LIN {X 0,Y 499.621,Z 974.079,A -85,B 0,C 180,E1 -11819.006,E2 -11819.006} C_VEL
LIN {X 0,Y 503.101,Z 958.378,A -85,B 0,C 180,E1 -11821.283,E2 -11821.283} C_VEL
LIN {X 0,Y 506.634,Z 942.412,A -85,B 0,C 180,E1 -11823.275,E2 -11823.275} C_VEL
LIN {X 0,Y 510.604,Z 924.617,A -85,B 0,C 180,E1 -11825.226,E2 -11825.226} C_VEL
LIN {X 0,Y 514.669,Z 905.302,A -85,B 0,C 180,E1 -11827.032,E2 -11827.032} C_VEL
LIN {X 0,Y 518.595,Z 886.147,A -85,B 0,C 180,E1 -11828.589,E2 -11828.589} C_VEL
LIN {X 0,Y 522.625,Z 864.682,A -85,B 0,C 180,E1 -11830.067,E2 -11830.067} C_VEL
LIN {X 0,Y 525.92,Z 845.573,A -85,B 0,C 180,E1 -11831.195,E2 -11831.195} C_VEL
LIN {X 0,Y 529.613,Z 821.59,A -85,B 0,C 180,E1 -11832.377,E2 -11832.377} C_VEL
LIN {X 0,Y 532.123,Z 802.454,A -85,B 0,C 180,E1 -11833.155,E2 -11833.155} C_VEL
LIN {X 0,Y 534.743,Z 779.457,A -85,B 0,C 180,E1 -11833.92,E2 -11833.92} C_VEL
LIN {X 0,Y 536.744,Z 755.79,A -85,B 0,C 180,E1 -11834.509,E2 -11834.509} C_VEL
LIN {X 0,Y 538.049,Z 733.759,A -85,B 0,C 180,E1 -11834.915,E2 -11834.915} C_VEL
LIN {X 0,Y 547.283,Z 482.875,A -85,B 0,C 180,E1 -11838.589,E2 -11838.589} C_VEL
LIN {X 0,Y 548.708,Z 441.821,A -85,B 0,C 180,E1 -11839.21,E2 -11839.21} C_VEL
LIN {X 0,Y 535.529,Z 420.602,A -85,B 0,C 180,E1 -11841.248,E2 -11841.248} C_VEL
LIN {X 0,Y 523.411,Z 403.652,A -85,B 0,C 180,E1 -11843.243,E2 -11843.243} C_VEL
LIN {X 0,Y 511.927,Z 388.487,A -85,B 0,C 180,E1 -11845.295,E2 -11845.295} C_VEL
LIN {X 0,Y 507.19,Z 382.618,A -85,B 0,C 180,E1 -11846.19,E2 -11846.19} C_VEL
LIN {X 0,Y 503.446,Z 377.826,A -85,B 0,C 180,E1 -11846.929,E2 -11846.929} C_VEL
LIN {X 0,Y 500.235,Z 374.018,A -85,B 0,C 180,E1 -11847.575,E2 -11847.575} C_VEL
LIN {X 0,Y 498.921,Z 372.158,A -85,B 0,C 180,E1 -11847.853,E2 -11847.853} C_VEL
LIN {X 0,Y 495.879,Z 368.896,A -85,B 0,C 180,E1 -11848.483,E2 -11848.483} C_VEL
LIN {X 0,Y 494.405,Z 366.407,A -85,B 0,C 180,E1 -11848.819,E2 -11848.819} C_VEL
LIN {X 0,Y 491.612,Z 364.144,A -85,B 0,C 180,E1 -11849.404,E2 -11849.404} C_VEL
LIN {X 0,Y 490.187,Z 361.183,A -85,B 0,C 180,E1 -11849.758,E2 -11849.758} C_VEL
LIN {X 0,Y 490,Z 360.194,A -85,B 0,C 180,E1 -11849.835,E2 -11849.835} C_VEL
LIN {X 0,Y 489.946,Z 360.203,A -85,B 0,C 180,E1 -11853.191,E2 -11853.191} C_VEL
LIN {X 0,Y 489.937,Z 360.203,A -85,B 0,C 180,E1 -11856.803,E2 -11856.803} C_VEL
LIN {X 0,Y 489.981,Z 360.199,A -85,B 0,C 180,E1 -11860.199,E2 -11860.199} C_VEL
LIN {X 0,Y 489.973,Z 360.196,A -85,B 0,C 180,E1 -11863.765,E2 -11863.765} C_VEL
LIN {X 0,Y 489.933,Z 360.192,A -85,B 0,C 180,E1 -11867.147,E2 -11867.147} C_VEL
LIN {X 0,Y 489.954,Z 360.179,A -85,B 0,C 180,E1 -11870.604,E2 -11870.604} C_VEL
LIN {X 0,Y 489.968,Z 360.177,A -85,B 0,C 180,E1 -11873.908,E2 -11873.908} C_VEL
LIN {X 0,Y 489.934,Z 360.192,A -85,B 0,C 180,E1 -11877.427,E2 -11877.427} C_VEL
LIN {X 0,Y 489.94,Z 360.201,A -85,B 0,C 180,E1 -11881.052,E2 -11881.052} C_VEL
LIN {X 0,Y 489.979,Z 360.194,A -85,B 0,C 180,E1 -11884.565,E2 -11884.565} C_VEL
LIN {X 0,Y 489.951,Z 360.18,A -85,B 0,C 180,E1 -11887.977,E2 -11887.977} C_VEL
LIN {X 0,Y 489.93,Z 360.176,A -85,B 0,C 180,E1 -11891.418,E2 -11891.418} C_VEL
LIN {X 0,Y 489.964,Z 360.175,A -85,B 0,C 180,E1 -11894.9,E2 -11894.9} C_VEL
LIN {X 0,Y 489.974,Z 360.182,A -85,B 0,C 180,E1 -11898.391,E2 -11898.391} C_VEL
LIN {X 0,Y 489.933,Z 360.199,A -85,B 0,C 180,E1 -11901.804,E2 -11901.804} C_VEL
LIN {X 0,Y 489.943,Z 360.201,A -85,B 0,C 180,E1 -11905.377,E2 -11905.377} C_VEL
LIN {X 0,Y 489.992,Z 360.197,A -85,B 0,C 180,E1 -11908.923,E2 -11908.923} C_VEL
LIN {X 0,Y 490.017,Z 360.424,A -85,B 0,C 180,E1 -11910.673,E2 -11910.673} C_VEL
LIN {X 0,Y 491.418,Z 363.93,A -85,B 0,C 180,E1 -11911.528,E2 -11911.528} C_VEL
LIN {X 0,Y 492.392,Z 365.741,A -85,B 0,C 180,E1 -11912.006,E2 -11912.006} C_VEL
LIN {X 0,Y 494.518,Z 369.645,A -85,B 0,C 180,E1 -11912.954,E2 -11912.954} C_VEL
LIN {X 0,Y 497.801,Z 374.223,A -85,B 0,C 180,E1 -11913.668,E2 -11913.668} C_VEL
LIN {X 0,Y 507.638,Z 387.39,A -85,B 0,C 180,E1 -11915.664,E2 -11915.664} C_VEL
LIN {X 0,Y 516.631,Z 399.971,A -85,B 0,C 180,E1 -11917.355,E2 -11917.355} C_VEL
LIN {X 0,Y 527.787,Z 416.461,A -85,B 0,C 180,E1 -11919.307,E2 -11919.307} C_VEL
LIN {X 0,Y 540.338,Z 436.58,A -85,B 0,C 180,E1 -11921.348,E2 -11921.348} C_VEL
LIN {X 0,Y 548.723,Z 451.311,A -85,B 0,C 180,E1 -11922.64,E2 -11922.64} C_VEL
LIN {X 0,Y 539.479,Z 702.482,A -85,B 0,C 180,E1 -11926.318,E2 -11926.318} C_VEL
LIN {X 0,Y 537.078,Z 765.181,A -85,B 0,C 180,E1 -11927.257,E2 -11927.257} C_VEL
LIN {X 0,Y 535.059,Z 790.28,A -85,B 0,C 180,E1 -11927.793,E2 -11927.793} C_VEL
LIN {X 0,Y 532.837,Z 811.473,A -85,B 0,C 180,E1 -11928.394,E2 -11928.394} C_VEL
LIN {X 0,Y 529.672,Z 836.124,A -85,B 0,C 180,E1 -11929.291,E2 -11929.291} C_VEL
LIN {X 0,Y 526.628,Z 856.667,A -85,B 0,C 180,E1 -11930.219,E2 -11930.219} C_VEL
LIN {X 0,Y 522.863,Z 879.253,A -85,B 0,C 180,E1 -11931.434,E2 -11931.434} C_VEL
LIN {X 0,Y 519.029,Z 900.032,A -85,B 0,C 180,E1 -11932.778,E2 -11932.778} C_VEL
LIN {X 0,Y 515.052,Z 920.507,A -85,B 0,C 180,E1 -11934.312,E2 -11934.312} C_VEL
LIN {X 0,Y 510.952,Z 940.064,A -85,B 0,C 180,E1 -11936.041,E2 -11936.041} C_VEL
LIN {X 0,Y 507.093,Z 958.257,A -85,B 0,C 180,E1 -11937.879,E2 -11937.879} C_VEL
LIN {X 0,Y 503.262,Z 975.902,A -85,B 0,C 180,E1 -11939.955,E2 -11939.955} C_VEL
LIN {X 0,Y 499.916,Z 991.806,A -85,B 0,C 180,E1 -11942.094,E2 -11942.094} C_VEL
LIN {X 0,Y 496.763,Z 1007.17,A -85,B 0,C 180,E1 -11944.485,E2 -11944.485} C_VEL
LIN {X 0,Y 494.443,Z 1019.312,A -85,B 0,C 180,E1 -11946.651,E2 -11946.651} C_VEL
LIN {X 0,Y 492.101,Z 1032.754,A -85,B 0,C 180,E1 -11949.42,E2 -11949.42} C_VEL
LIN {X 0,Y 490.58,Z 1042.696,A -85,B 0,C 180,E1 -11951.83,E2 -11951.83} C_VEL
LIN {X 0,Y 489.408,Z 1052.094,A -85,B 0,C 180,E1 -11954.476,E2 -11954.476} C_VEL
LIN {X 0,Y 488.611,Z 1060.001,A -85,B 0,C 180,E1 -11957.232,E2 -11957.232} C_VEL
LIN {X 0,Y 488.21,Z 1065.616,A -85,B 0,C 180,E1 -11959.617,E2 -11959.617} C_VEL
LIN {X 0,Y 487.988,Z 1070.959,A -85,B 0,C 180,E1 -11962.583,E2 -11962.583} C_VEL
LIN {X 0,Y 487.94,Z 1074.004,A -85,B 0,C 180,E1 -11965.063,E2 -11965.063} C_VEL
LIN {X 0,Y 487.927,Z 1075.86,A -85,B 0,C 180,E1 -11967.534,E2 -11967.534} C_VEL
LIN {X 0,Y 487.924,Z 1076.467,A -85,B 0,C 180,E1 -11970.352,E2 -11970.352} C_VEL
LIN {X 0,Y 487.93,Z 1075.637,A -85,B 0,C 180,E1 -11972.819,E2 -11972.819} C_VEL
LIN {X 0,Y 487.941,Z 1073.628,A -85,B 0,C 180,E1 -11975.291,E2 -11975.291} C_VEL
LIN {X 0,Y 488.035,Z 1069.53,A -85,B 0,C 180,E1 -11978.279,E2 -11978.279} C_VEL
LIN {X 0,Y 488.264,Z 1064.748,A -85,B 0,C 180,E1 -11980.74,E2 -11980.74} C_VEL
LIN {X 0,Y 488.784,Z 1058.014,A -85,B 0,C 180,E1 -11983.486,E2 -11983.486} C_VEL
LIN {X 0,Y 489.667,Z 1049.398,A -85,B 0,C 180,E1 -11986.245,E2 -11986.245} C_VEL
LIN {X 0,Y 490.902,Z 1040.057,A -85,B 0,C 180,E1 -11988.773,E2 -11988.773} C_VEL
LIN {X 0,Y 492.69,Z 1028.406,A -85,B 0,C 180,E1 -11991.426,E2 -11991.426} C_VEL
LIN {X 0,Y 494.724,Z 1016.75,A -85,B 0,C 180,E1 -11993.716,E2 -11993.716} C_VEL
LIN {X 0,Y 497.688,Z 1001.146,A -85,B 0,C 180,E1 -11996.36,E2 -11996.36} C_VEL
LIN {X 0,Y 500.61,Z 986.526,A -85,B 0,C 180,E1 -11998.498,E2 -11998.498} C_VEL
LIN {X 0,Y 504.41,Z 968.165,A -85,B 0,C 180,E1 -12000.825,E2 -12000.825} C_VEL
LIN {X 0,Y 507.711,Z 952.169,A -85,B 0,C 180,E1 -12002.584,E2 -12002.584} C_VEL
LIN {X 0,Y 511.658,Z 932.877,A -85,B 0,C 180,E1 -12004.443,E2 -12004.443} C_VEL
LIN {X 0,Y 515.488,Z 913.172,A -85,B 0,C 180,E1 -12006.065,E2 -12006.065} C_VEL
LIN {X 0,Y 519.375,Z 892.502,A -85,B 0,C 180,E1 -12007.54,E2 -12007.54} C_VEL
LIN {X 0,Y 522.872,Z 871.802,A -85,B 0,C 180,E1 -12008.782,E2 -12008.782} C_VEL
LIN {X 0,Y 525.902,Z 852.464,A -85,B 0,C 180,E1 -12009.776,E2 -12009.776} C_VEL
LIN {X 0,Y 529.266,Z 827.978,A -85,B 0,C 180,E1 -12010.818,E2 -12010.818} C_VEL
LIN {X 0,Y 531.66,Z 807.467,A -85,B 0,C 180,E1 -12011.517,E2 -12011.517} C_VEL
LIN {X 0,Y 533.992,Z 783.772,A -85,B 0,C 180,E1 -12012.157,E2 -12012.157} C_VEL
LIN {X 0,Y 535.574,Z 759.261,A -85,B 0,C 180,E1 -12012.627,E2 -12012.627} C_VEL
LIN {X 0,Y 543.706,Z 523.272,A -85,B 0,C 180,E1 -12016.069,E2 -12016.069} C_VEL
LIN {X 0,Y 546.171,Z 449.822,A -85,B 0,C 180,E1 -12017.16,E2 -12017.16} C_VEL
LIN {X 0,Y 533.572,Z 427.973,A -85,B 0,C 180,E1 -12019.013,E2 -12019.013} C_VEL
LIN {X 0,Y 520.585,Z 407.244,A -85,B 0,C 180,E1 -12021.056,E2 -12021.056} C_VEL
LIN {X 0,Y 507.929,Z 388.602,A -85,B 0,C 180,E1 -12023.206,E2 -12023.206} C_VEL
LIN {X 0,Y 497.103,Z 373.702,A -85,B 0,C 180,E1 -12025.198,E2 -12025.198} C_VEL
LIN {X 0,Y 494.207,Z 369.566,A -85,B 0,C 180,E1 -12025.774,E2 -12025.774} C_VEL
LIN {X 0,Y 492.163,Z 365.3,A -85,B 0,C 180,E1 -12026.733,E2 -12026.733} C_VEL
LIN {X 0,Y 489.994,Z 360.56,A -85,B 0,C 180,E1 -12027.818,E2 -12027.818} C_VEL
LIN {X 0,Y 489.934,Z 360.191,A -85,B 0,C 180,E1 -12027.952,E2 -12027.952} C_VEL
LIN {X 0,Y 489.991,Z 360.186,A -85,B 0,C 180,E1 -12031.344,E2 -12031.344} C_VEL
LIN {X 0,Y 489.963,Z 360.198,A -85,B 0,C 180,E1 -12034.882,E2 -12034.882} C_VEL
LIN {X 0,Y 489.931,Z 360.197,A -85,B 0,C 180,E1 -12038.321,E2 -12038.321} C_VEL
LIN {X 0,Y 489.956,Z 360.176,A -85,B 0,C 180,E1 -12041.806,E2 -12041.806} C_VEL
LIN {X 0,Y 489.99,Z 360.167,A -85,B 0,C 180,E1 -12045.343,E2 -12045.343} C_VEL
LIN {X 0,Y 489.941,Z 360.196,A -85,B 0,C 180,E1 -12048.821,E2 -12048.821} C_VEL
LIN {X 0,Y 489.934,Z 360.198,A -85,B 0,C 180,E1 -12052.377,E2 -12052.377} C_VEL
LIN {X 0,Y 489.975,Z 360.165,A -85,B 0,C 180,E1 -12055.787,E2 -12055.787} C_VEL
LIN {X 0,Y 489.962,Z 360.184,A -85,B 0,C 180,E1 -12059.298,E2 -12059.298} C_VEL
LIN {X 0,Y 489.934,Z 360.201,A -85,B 0,C 180,E1 -12062.808,E2 -12062.808} C_VEL
LIN {X 0,Y 489.946,Z 360.169,A -85,B 0,C 180,E1 -12066.344,E2 -12066.344} C_VEL
LIN {X 0,Y 489.983,Z 360.18,A -85,B 0,C 180,E1 -12069.752,E2 -12069.752} C_VEL
LIN {X 0,Y 489.942,Z 360.199,A -85,B 0,C 180,E1 -12073.226,E2 -12073.226} C_VEL
LIN {X 0,Y 489.934,Z 360.176,A -85,B 0,C 180,E1 -12076.846,E2 -12076.846} C_VEL
LIN {X 0,Y 489.973,Z 360.171,A -85,B 0,C 180,E1 -12080.299,E2 -12080.299} C_VEL
LIN {X 0,Y 489.964,Z 360.195,A -85,B 0,C 180,E1 -12083.705,E2 -12083.705} C_VEL
LIN {X 0,Y 489.94,Z 360.202,A -85,B 0,C 180,E1 -12087.203,E2 -12087.203} C_VEL
LIN {X 0,Y 489.957,Z 360.186,A -85,B 0,C 180,E1 -12090.677,E2 -12090.677} C_VEL
LIN {X 0,Y 489.984,Z 360.179,A -85,B 0,C 180,E1 -12094.138,E2 -12094.138} C_VEL
LIN {X 0,Y 489.958,Z 360.256,A -85,B 0,C 180,E1 -12095.709,E2 -12095.709} C_VEL
LIN {X 0,Y 491.007,Z 363.245,A -85,B 0,C 180,E1 -12095.962,E2 -12095.962} C_VEL
LIN {X 0,Y 493.4,Z 365.788,A -85,B 0,C 180,E1 -12096.425,E2 -12096.425} C_VEL
LIN {X 0,Y 494.526,Z 366.796,A -85,B 0,C 180,E1 -12096.635,E2 -12096.635} C_VEL
LIN {X 0,Y 496.989,Z 370.604,A -85,B 0,C 180,E1 -12097.126,E2 -12097.126} C_VEL
LIN {X 0,Y 499.262,Z 372.917,A -85,B 0,C 180,E1 -12097.542,E2 -12097.542} C_VEL
LIN {X 0,Y 502.564,Z 377.233,A -85,B 0,C 180,E1 -12098.153,E2 -12098.153} C_VEL
LIN {X 0,Y 512.006,Z 389.56,A -85,B 0,C 180,E1 -12099.815,E2 -12099.815} C_VEL
LIN {X 0,Y 523.641,Z 405.343,A -85,B 0,C 180,E1 -12101.718,E2 -12101.718} C_VEL
LIN {X 0,Y 534.992,Z 421.994,A -85,B 0,C 180,E1 -12103.455,E2 -12103.455} C_VEL
LIN {X 0,Y 546.448,Z 441.202,A -85,B 0,C 180,E1 -12105.128,E2 -12105.128} C_VEL
LIN {X 0,Y 537.807,Z 687.67,A -85,B 0,C 180,E1 -12108.714,E2 -12108.714} C_VEL
LIN {X 0,Y 535.684,Z 744.725,A -85,B 0,C 180,E1 -12109.568,E2 -12109.568} C_VEL
LIN {X 0,Y 533.884,Z 769.233,A -85,B 0,C 180,E1 -12110.108,E2 -12110.108} C_VEL
LIN {X 0,Y 531.773,Z 791.218,A -85,B 0,C 180,E1 -12110.75,E2 -12110.75} C_VEL
LIN {X 0,Y 528.953,Z 814.971,A -85,B 0,C 180,E1 -12111.639,E2 -12111.639} C_VEL
LIN {X 0,Y 526.187,Z 834.834,A -85,B 0,C 180,E1 -12112.549,E2 -12112.549} C_VEL
LIN {X 0,Y 522.677,Z 857.192,A -85,B 0,C 180,E1 -12113.763,E2 -12113.763} C_VEL
LIN {X 0,Y 519.054,Z 877.695,A -85,B 0,C 180,E1 -12115.101,E2 -12115.101} C_VEL
LIN {X 0,Y 515.255,Z 897.885,A -85,B 0,C 180,E1 -12116.623,E2 -12116.623} C_VEL
LIN {X 0,Y 511.312,Z 917.088,A -85,B 0,C 180,E1 -12118.328,E2 -12118.328} C_VEL
LIN {X 0,Y 510.97,Z 918.726,A -85,B 0,C 180,E1 -12118.484,E2 -12118.484} C_VEL
LIN {X 0,Y 508.908,Z 924.702,A -85,B 0,C 180,E1 -12118.999,E2 -12118.999} C_VEL
LIN {X 0,Y 500.503,Z 939.528,A -85,B 0,C 180,E1 -12120.219,E2 -12120.219} C_VEL
LIN {X 0,Y 498.41,Z 944.959,A -85,B 0,C 180,E1 -12120.796,E2 -12120.796} C_VEL
LIN {X 0,Y 494.435,Z 962.729,A -85,B 0,C 180,E1 -12123.105,E2 -12123.105} C_VEL
LIN {X 0,Y 491.323,Z 976.784,A -85,B 0,C 180,E1 -12125.214,E2 -12125.214} C_VEL
LIN {X 0,Y 488.087,Z 992.002,A -85,B 0,C 180,E1 -12127.856,E2 -12127.856} C_VEL
LIN {X 0,Y 485.71,Z 1003.891,A -85,B 0,C 180,E1 -12130.269,E2 -12130.269} C_VEL
LIN {X 0,Y 483.54,Z 1016.07,A -85,B 0,C 180,E1 -12133.172,E2 -12133.172} C_VEL
LIN {X 0,Y 482.208,Z 1024.593,A -85,B 0,C 180,E1 -12135.592,E2 -12135.592} C_VEL
LIN {X 0,Y 481.157,Z 1032.862,A -85,B 0,C 180,E1 -12138.371,E2 -12138.371} C_VEL
LIN {X 0,Y 480.498,Z 1039.328,A -85,B 0,C 180,E1 -12141.142,E2 -12141.142} C_VEL
LIN {X 0,Y 480.163,Z 1043.981,A -85,B 0,C 180,E1 -12143.664,E2 -12143.664} C_VEL
LIN {X 0,Y 479.987,Z 1047.874,A -85,B 0,C 180,E1 -12146.656,E2 -12146.656} C_VEL
LIN {X 0,Y 479.945,Z 1049.749,A -85,B 0,C 180,E1 -12149.045,E2 -12149.045} C_VEL
LIN {X 0,Y 479.923,Z 1050.584,A -85,B 0,C 180,E1 -12151.433,E2 -12151.433} C_VEL
LIN {X 0,Y 479.94,Z 1050.138,A -85,B 0,C 180,E1 -12154.421,E2 -12154.421} C_VEL
LIN {X 0,Y 479.981,Z 1048.405,A -85,B 0,C 180,E1 -12156.94,E2 -12156.94} C_VEL
LIN {X 0,Y 480.088,Z 1045.678,A -85,B 0,C 180,E1 -12159.349,E2 -12159.349} C_VEL
LIN {X 0,Y 480.404,Z 1040.694,A -85,B 0,C 180,E1 -12162.379,E2 -12162.379} C_VEL
LIN {X 0,Y 480.947,Z 1035.03,A -85,B 0,C 180,E1 -12164.939,E2 -12164.939} C_VEL
LIN {X 0,Y 481.928,Z 1027.365,A -85,B 0,C 180,E1 -12167.763,E2 -12167.763} C_VEL
LIN {X 0,Y 483.383,Z 1017.776,A -85,B 0,C 180,E1 -12170.588,E2 -12170.588} C_VEL
LIN {X 0,Y 485.367,Z 1006.968,A -85,B 0,C 180,E1 -12173.299,E2 -12173.299} C_VEL
LIN {X 0,Y 487.847,Z 994.643,A -85,B 0,C 180,E1 -12175.885,E2 -12175.885} C_VEL
LIN {X 0,Y 490.638,Z 981.902,A -85,B 0,C 180,E1 -12178.216,E2 -12178.216} C_VEL
LIN {X 0,Y 494.168,Z 966.354,A -85,B 0,C 180,E1 -12180.657,E2 -12180.657} C_VEL
LIN {X 0,Y 497.539,Z 951.848,A -85,B 0,C 180,E1 -12182.642,E2 -12182.642} C_VEL
LIN {X 0,Y 501.913,Z 933.015,A -85,B 0,C 180,E1 -12184.872,E2 -12184.872} C_VEL
LIN {X 0,Y 505.593,Z 916.81,A -85,B 0,C 180,E1 -12186.532,E2 -12186.532} C_VEL
LIN {X 0,Y 509.926,Z 897.147,A -85,B 0,C 180,E1 -12188.289,E2 -12188.289} C_VEL
LIN {X 0,Y 513.894,Z 877.606,A -85,B 0,C 180,E1 -12189.775,E2 -12189.775} C_VEL
LIN {X 0,Y 517.938,Z 856.354,A -85,B 0,C 180,E1 -12191.171,E2 -12191.171} C_VEL
LIN {X 0,Y 521.615,Z 834.431,A -85,B 0,C 180,E1 -12192.361,E2 -12192.361} C_VEL
LIN {X 0,Y 524.717,Z 813.622,A -85,B 0,C 180,E1 -12193.315,E2 -12193.315} C_VEL
LIN {X 0,Y 527.783,Z 789.004,A -85,B 0,C 180,E1 -12194.22,E2 -12194.22} C_VEL
LIN {X 0,Y 530.012,Z 767.069,A -85,B 0,C 180,E1 -12194.85,E2 -12194.85} C_VEL
LIN {X 0,Y 531.932,Z 740.911,A -85,B 0,C 180,E1 -12195.396,E2 -12195.396} C_VEL
LIN {X 0,Y 540.8,Z 510.38,A -85,B 0,C 180,E1 -12198.811,E2 -12198.811} C_VEL
LIN {X 0,Y 543.236,Z 445.431,A -85,B 0,C 180,E1 -12199.789,E2 -12199.789} C_VEL
LIN {X 0,Y 530.888,Z 425.495,A -85,B 0,C 180,E1 -12201.752,E2 -12201.752} C_VEL
LIN {X 0,Y 519.483,Z 409.528,A -85,B 0,C 180,E1 -12203.676,E2 -12203.676} C_VEL
LIN {X 0,Y 508.649,Z 395.076,A -85,B 0,C 180,E1 -12205.655,E2 -12205.655} C_VEL
LIN {X 0,Y 503.459,Z 388.623,A -85,B 0,C 180,E1 -12206.658,E2 -12206.658} C_VEL
LIN {X 0,Y 500.253,Z 384.501,A -85,B 0,C 180,E1 -12207.305,E2 -12207.305} C_VEL
LIN {X 0,Y 496.742,Z 380.013,A -85,B 0,C 180,E1 -12208.035,E2 -12208.035} C_VEL
LIN {X 0,Y 492.563,Z 375.092,A -85,B 0,C 180,E1 -12208.927,E2 -12208.927} C_VEL
LIN {X 0,Y 491.539,Z 373.531,A -85,B 0,C 180,E1 -12209.161,E2 -12209.161} C_VEL
LIN {X 0,Y 488.465,Z 370.552,A -85,B 0,C 180,E1 -12209.832,E2 -12209.832} C_VEL
LIN {X 0,Y 486.735,Z 367.519,A -85,B 0,C 180,E1 -12210.257,E2 -12210.257} C_VEL
LIN {X 0,Y 483.812,Z 365.336,A -85,B 0,C 180,E1 -12210.909,E2 -12210.909} C_VEL
LIN {X 0,Y 482.264,Z 362.395,A -85,B 0,C 180,E1 -12211.316,E2 -12211.316} C_VEL
LIN {X 0,Y 482.022,Z 361.171,A -85,B 0,C 180,E1 -12211.425,E2 -12211.425} C_VEL
LIN {X 0,Y 481.997,Z 361.171,A -85,B 0,C 180,E1 -12214.963,E2 -12214.963} C_VEL
LIN {X 0,Y 482.013,Z 361.168,A -85,B 0,C 180,E1 -12218.459,E2 -12218.459} C_VEL
LIN {X 0,Y 482.042,Z 361.165,A -85,B 0,C 180,E1 -12221.872,E2 -12221.872} C_VEL
LIN {X 0,Y 481.999,Z 361.173,A -85,B 0,C 180,E1 -12225.34,E2 -12225.34} C_VEL
LIN {X 0,Y 482,Z 361.182,A -85,B 0,C 180,E1 -12228.879,E2 -12228.879} C_VEL
LIN {X 0,Y 482.043,Z 361.186,A -85,B 0,C 180,E1 -12232.371,E2 -12232.371} C_VEL
LIN {X 0,Y 482.029,Z 361.182,A -85,B 0,C 180,E1 -12235.956,E2 -12235.956} C_VEL
LIN {X 0,Y 481.993,Z 361.172,A -85,B 0,C 180,E1 -12239.406,E2 -12239.406} C_VEL
LIN {X 0,Y 482.002,Z 361.165,A -85,B 0,C 180,E1 -12242.973,E2 -12242.973} C_VEL
LIN {X 0,Y 482.05,Z 361.162,A -85,B 0,C 180,E1 -12246.504,E2 -12246.504} C_VEL
LIN {X 0,Y 482.015,Z 361.178,A -85,B 0,C 180,E1 -12250.035,E2 -12250.035} C_VEL
LIN {X 0,Y 481.994,Z 361.191,A -85,B 0,C 180,E1 -12253.557,E2 -12253.557} C_VEL
LIN {X 0,Y 482.02,Z 361.181,A -85,B 0,C 180,E1 -12257.007,E2 -12257.007} C_VEL
LIN {X 0,Y 482.042,Z 361.168,A -85,B 0,C 180,E1 -12260.521,E2 -12260.521} C_VEL
LIN {X 0,Y 481.994,Z 361.168,A -85,B 0,C 180,E1 -12263.862,E2 -12263.862} C_VEL
LIN {X 0,Y 482.002,Z 361.168,A -85,B 0,C 180,E1 -12267.421,E2 -12267.421} C_VEL
LIN {X 0,Y 482.039,Z 361.318,A -85,B 0,C 180,E1 -12269.208,E2 -12269.208} C_VEL
LIN {X 0,Y 483.265,Z 364.613,A -85,B 0,C 180,E1 -12270.047,E2 -12270.047} C_VEL
LIN {X 0,Y 484.518,Z 366.617,A -85,B 0,C 180,E1 -12270.646,E2 -12270.646} C_VEL
LIN {X 0,Y 485.699,Z 369.227,A -85,B 0,C 180,E1 -12271.251,E2 -12271.251} C_VEL
LIN {X 0,Y 491.205,Z 375.925,A -85,B 0,C 180,E1 -12272.507,E2 -12272.507} C_VEL
LIN {X 0,Y 495.053,Z 381.243,A -85,B 0,C 180,E1 -12273.359,E2 -12273.359} C_VEL
LIN {X 0,Y 506.429,Z 396.637,A -85,B 0,C 180,E1 -12275.693,E2 -12275.693} C_VEL
LIN {X 0,Y 516.502,Z 411.273,A -85,B 0,C 180,E1 -12277.593,E2 -12277.593} C_VEL
LIN {X 0,Y 527.061,Z 427.405,A -85,B 0,C 180,E1 -12279.442,E2 -12279.442} C_VEL
LIN {X 0,Y 538.473,Z 446.211,A -85,B 0,C 180,E1 -12281.31,E2 -12281.31} C_VEL
LIN {X 0,Y 543.243,Z 454.931,A -85,B 0,C 180,E1 -12282.064,E2 -12282.064} C_VEL
LIN {X 0,Y 533.685,Z 704.84,A -85,B 0,C 180,E1 -12285.751,E2 -12285.751} C_VEL
LIN {X 0,Y 531.274,Z 765.234,A -85,B 0,C 180,E1 -12286.664,E2 -12286.664} C_VEL
LIN {X 0,Y 529.199,Z 790.162,A -85,B 0,C 180,E1 -12287.201,E2 -12287.201} C_VEL
LIN {X 0,Y 526.93,Z 811.121,A -85,B 0,C 180,E1 -12287.798,E2 -12287.798} C_VEL
LIN {X 0,Y 523.593,Z 836.206,A -85,B 0,C 180,E1 -12288.716,E2 -12288.716} C_VEL
LIN {X 0,Y 520.443,Z 856.712,A -85,B 0,C 180,E1 -12289.65,E2 -12289.65} C_VEL
LIN {X 0,Y 516.41,Z 879.898,A -85,B 0,C 180,E1 -12290.912,E2 -12290.912} C_VEL
LIN {X 0,Y 512.556,Z 900,A -85,B 0,C 180,E1 -12292.226,E2 -12292.226} C_VEL
LIN {X 0,Y 508.269,Z 921.119,A -85,B 0,C 180,E1 -12293.831,E2 -12293.831} C_VEL
LIN {X 0,Y 504.207,Z 939.745,A -85,B 0,C 180,E1 -12295.496,E2 -12295.496} C_VEL
LIN {X 0,Y 500.318,Z 957.3,A -85,B 0,C 180,E1 -12297.286,E2 -12297.286} C_VEL
LIN {X 0,Y 496.118,Z 975.783,A -85,B 0,C 180,E1 -12299.477,E2 -12299.477} C_VEL
LIN {X 0,Y 492.794,Z 990.826,A -85,B 0,C 180,E1 -12301.522,E2 -12301.522} C_VEL
LIN {X 0,Y 489.298,Z 1007.022,A -85,B 0,C 180,E1 -12304.067,E2 -12304.067} C_VEL
LIN {X 0,Y 486.851,Z 1019.146,A -85,B 0,C 180,E1 -12306.263,E2 -12306.263} C_VEL
LIN {X 0,Y 484.368,Z 1032.585,A -85,B 0,C 180,E1 -12309.076,E2 -12309.076} C_VEL
LIN {X 0,Y 482.744,Z 1042.645,A -85,B 0,C 180,E1 -12311.558,E2 -12311.558} C_VEL
LIN {X 0,Y 481.465,Z 1052.283,A -85,B 0,C 180,E1 -12314.337,E2 -12314.337} C_VEL
LIN {X 0,Y 480.662,Z 1059.81,A -85,B 0,C 180,E1 -12317.017,E2 -12317.017} C_VEL
LIN {X 0,Y 480.236,Z 1065.421,A -85,B 0,C 180,E1 -12319.442,E2 -12319.442} C_VEL
LIN {X 0,Y 479.987,Z 1070.757,A -85,B 0,C 180,E1 -12322.459,E2 -12322.459} C_VEL
LIN {X 0,Y 479.941,Z 1073.798,A -85,B 0,C 180,E1 -12324.98,E2 -12324.98} C_VEL
LIN {X 0,Y 479.929,Z 1075.652,A -85,B 0,C 180,E1 -12327.492,E2 -12327.492} C_VEL
LIN {X 0,Y 479.927,Z 1076.252,A -85,B 0,C 180,E1 -12330.358,E2 -12330.358} C_VEL
LIN {X 0,Y 479.932,Z 1075.418,A -85,B 0,C 180,E1 -12332.866,E2 -12332.866} C_VEL
LIN {X 0,Y 479.942,Z 1073.521,A -85,B 0,C 180,E1 -12335.26,E2 -12335.26} C_VEL
LIN {X 0,Y 480.021,Z 1069.777,A -85,B 0,C 180,E1 -12338.143,E2 -12338.143} C_VEL
LIN {X 0,Y 480.272,Z 1064.769,A -85,B 0,C 180,E1 -12340.799,E2 -12340.799} C_VEL
LIN {X 0,Y 480.779,Z 1058.388,A -85,B 0,C 180,E1 -12343.47,E2 -12343.47} C_VEL
LIN {X 0,Y 481.734,Z 1049.553,A -85,B 0,C 180,E1 -12346.396,E2 -12346.396} C_VEL
LIN {X 0,Y 482.981,Z 1040.525,A -85,B 0,C 180,E1 -12348.896,E2 -12348.896} C_VEL
LIN {X 0,Y 484.994,Z 1028.127,A -85,B 0,C 180,E1 -12351.783,E2 -12351.783} C_VEL
LIN {X 0,Y 487.133,Z 1016.462,A -85,B 0,C 180,E1 -12354.109,E2 -12354.109} C_VEL
LIN {X 0,Y 490.255,Z 1000.843,A -85,B 0,C 180,E1 -12356.791,E2 -12356.791} C_VEL
LIN {X 0,Y 493.157,Z 986.966,A -85,B 0,C 180,E1 -12358.852,E2 -12358.852} C_VEL
LIN {X 0,Y 496.98,Z 969.373,A -85,B 0,C 180,E1 -12361.136,E2 -12361.136} C_VEL
LIN {X 0,Y 500.64,Z 952.33,A -85,B 0,C 180,E1 -12363.041,E2 -12363.041} C_VEL
LIN {X 0,Y 504.753,Z 933.076,A -85,B 0,C 180,E1 -12364.924,E2 -12364.924} C_VEL
LIN {X 0,Y 508.709,Z 913.527,A -85,B 0,C 180,E1 -12366.553,E2 -12366.553} C_VEL
LIN {X 0,Y 512.731,Z 892.926,A -85,B 0,C 180,E1 -12368.042,E2 -12368.042} C_VEL
LIN {X 0,Y 516.511,Z 871.435,A -85,B 0,C 180,E1 -12369.345,E2 -12369.345} C_VEL
LIN {X 0,Y 519.735,Z 851.531,A -85,B 0,C 180,E1 -12370.373,E2 -12370.373} C_VEL
LIN {X 0,Y 523.141,Z 827.416,A -85,B 0,C 180,E1 -12371.4,E2 -12371.4} C_VEL
LIN {X 0,Y 525.598,Z 807.062,A -85,B 0,C 180,E1 -12372.096,E2 -12372.096} C_VEL
LIN {X 0,Y 527.992,Z 783.427,A -85,B 0,C 180,E1 -12372.736,E2 -12372.736} C_VEL
LIN {X 0,Y 529.62,Z 758.915,A -85,B 0,C 180,E1 -12373.208,E2 -12373.208} C_VEL
LIN {X 0,Y 538.1,Z 522.435,A -85,B 0,C 180,E1 -12376.686,E2 -12376.686} C_VEL
LIN {X 0,Y 540.511,Z 453.255,A -85,B 0,C 180,E1 -12377.722,E2 -12377.722} C_VEL
LIN {X 0,Y 528.792,Z 432.769,A -85,B 0,C 180,E1 -12379.494,E2 -12379.494} C_VEL
LIN {X 0,Y 515.955,Z 412.163,A -85,B 0,C 180,E1 -12381.567,E2 -12381.567} C_VEL
LIN {X 0,Y 504.122,Z 394.665,A -85,B 0,C 180,E1 -12383.626,E2 -12383.626} C_VEL
LIN {X 0,Y 493.941,Z 380.422,A -85,B 0,C 180,E1 -12385.542,E2 -12385.542} C_VEL
LIN {X 0,Y 489.755,Z 374.884,A -85,B 0,C 180,E1 -12386.373,E2 -12386.373} C_VEL
LIN {X 0,Y 485.508,Z 369.065,A -85,B 0,C 180,E1 -12387.275,E2 -12387.275} C_VEL
LIN {X 0,Y 483.704,Z 365.21,A -85,B 0,C 180,E1 -12388.188,E2 -12388.188} C_VEL
LIN {X 0,Y 482.252,Z 362.279,A -85,B 0,C 180,E1 -12388.917,E2 -12388.917} C_VEL
LIN {X 0,Y 482.057,Z 361.159,A -85,B 0,C 180,E1 -12389.181,E2 -12389.181} C_VEL
LIN {X 0,Y 482.002,Z 361.162,A -85,B 0,C 180,E1 -12392.606,E2 -12392.606} C_VEL
LIN {X 0,Y 481.992,Z 361.164,A -85,B 0,C 180,E1 -12396.185,E2 -12396.185} C_VEL
LIN {X 0,Y 482.029,Z 361.175,A -85,B 0,C 180,E1 -12399.652,E2 -12399.652} C_VEL
LIN {X 0,Y 482.042,Z 361.186,A -85,B 0,C 180,E1 -12403.242,E2 -12403.242} C_VEL
LIN {X 0,Y 481.996,Z 361.17,A -85,B 0,C 180,E1 -12406.687,E2 -12406.687} C_VEL
LIN {X 0,Y 481.994,Z 361.158,A -85,B 0,C 180,E1 -12410.326,E2 -12410.326} C_VEL
LIN {X 0,Y 482.038,Z 361.178,A -85,B 0,C 180,E1 -12413.808,E2 -12413.808} C_VEL
LIN {X 0,Y 482.031,Z 361.179,A -85,B 0,C 180,E1 -12417.384,E2 -12417.384} C_VEL
LIN {X 0,Y 481.991,Z 361.155,A -85,B 0,C 180,E1 -12420.832,E2 -12420.832} C_VEL
LIN {X 0,Y 482.005,Z 361.18,A -85,B 0,C 180,E1 -12424.402,E2 -12424.402} C_VEL
LIN {X 0,Y 482.055,Z 361.176,A -85,B 0,C 180,E1 -12427.868,E2 -12427.868} C_VEL
LIN {X 0,Y 482.018,Z 361.154,A -85,B 0,C 180,E1 -12431.487,E2 -12431.487} C_VEL
LIN {X 0,Y 481.995,Z 361.175,A -85,B 0,C 180,E1 -12434.906,E2 -12434.906} C_VEL
LIN {X 0,Y 482.028,Z 361.188,A -85,B 0,C 180,E1 -12438.379,E2 -12438.379} C_VEL
LIN {X 0,Y 482.055,Z 361.164,A -85,B 0,C 180,E1 -12442.001,E2 -12442.001} C_VEL
LIN {X 0,Y 482.009,Z 361.16,A -85,B 0,C 180,E1 -12445.562,E2 -12445.562} C_VEL
LIN {X 0,Y 482,Z 361.166,A -85,B 0,C 180,E1 -12449.04,E2 -12449.04} C_VEL
LIN {X 0,Y 482.038,Z 361.169,A -85,B 0,C 180,E1 -12452.496,E2 -12452.496} C_VEL
LIN {X 0,Y 482.072,Z 361.362,A -85,B 0,C 180,E1 -12454.345,E2 -12454.345} C_VEL
LIN {X 0,Y 483.137,Z 364.357,A -85,B 0,C 180,E1 -12454.618,E2 -12454.618} C_VEL
LIN {X 0,Y 485.642,Z 366.951,A -85,B 0,C 180,E1 -12455.132,E2 -12455.132} C_VEL
LIN {X 0,Y 486.744,Z 367.867,A -85,B 0,C 180,E1 -12455.349,E2 -12455.349} C_VEL
LIN {X 0,Y 489.116,Z 371.544,A -85,B 0,C 180,E1 -12455.852,E2 -12455.852} C_VEL
LIN {X 0,Y 491.447,Z 373.923,A -85,B 0,C 180,E1 -12456.304,E2 -12456.304} C_VEL
LIN {X 0,Y 494.642,Z 378.163,A -85,B 0,C 180,E1 -12456.933,E2 -12456.933} C_VEL
LIN {X 0,Y 496.343,Z 380.199,A -85,B 0,C 180,E1 -12457.255,E2 -12457.255} C_VEL
LIN {X 0,Y 501.344,Z 386.76,A -85,B 0,C 180,E1 -12458.19,E2 -12458.19} C_VEL
LIN {X 0,Y 505.654,Z 392.322,A -85,B 0,C 180,E1 -12458.963,E2 -12458.963} C_VEL
LIN {X 0,Y 515.74,Z 405.857,A -85,B 0,C 180,E1 -12460.686,E2 -12460.686} C_VEL
LIN {X 0,Y 527.75,Z 423.031,A -85,B 0,C 180,E1 -12462.599,E2 -12462.599} C_VEL
LIN {X 0,Y 539.534,Z 442.323,A -85,B 0,C 180,E1 -12464.377,E2 -12464.377} C_VEL
LIN {X 0,Y 540.795,Z 444.867,A -85,B 0,C 180,E1 -12464.568,E2 -12464.568} C_VEL
LIN {X 0,Y 531.788,Z 692,A -85,B 0,C 180,E1 -12468.192,E2 -12468.192} C_VEL
LIN {X 0,Y 529.701,Z 745.554,A -85,B 0,C 180,E1 -12469.003,E2 -12469.003} C_VEL
LIN {X 0,Y 527.831,Z 769.887,A -85,B 0,C 180,E1 -12469.548,E2 -12469.548} C_VEL
LIN {X 0,Y 525.596,Z 792.386,A -85,B 0,C 180,E1 -12470.213,E2 -12470.213} C_VEL
LIN {X 0,Y 522.608,Z 816.404,A -85,B 0,C 180,E1 -12471.13,E2 -12471.13} C_VEL
LIN {X 0,Y 519.646,Z 836.867,A -85,B 0,C 180,E1 -12472.084,E2 -12472.084} C_VEL
LIN {X 0,Y 515.736,Z 860.378,A -85,B 0,C 180,E1 -12473.404,E2 -12473.404} C_VEL
LIN {X 0,Y 512.213,Z 879.579,A -85,B 0,C 180,E1 -12474.685,E2 -12474.685} C_VEL
LIN {X 0,Y 507.952,Z 900.99,A -85,B 0,C 180,E1 -12476.35,E2 -12476.35} C_VEL
LIN {X 0,Y 504.181,Z 918.716,A -85,B 0,C 180,E1 -12477.96,E2 -12477.96} C_VEL
LIN {X 0,Y 500.171,Z 937.19,A -85,B 0,C 180,E1 -12479.883,E2 -12479.883} C_VEL
LIN {X 0,Y 498.41,Z 944.959,A -85,B 0,C 180,E1 -12480.796,E2 -12480.796} C_VEL
LIN {X 0,Y 496.317,Z 950.385,A -85,B 0,C 180,E1 -12481.393,E2 -12481.393} C_VEL
LIN {X 0,Y 487.897,Z 963.83,A -85,B 0,C 180,E1 -12482.837,E2 -12482.837} C_VEL
LIN {X 0,Y 485.877,Z 968.772,A -85,B 0,C 180,E1 -12483.495,E2 -12483.495} C_VEL
LIN {X 0,Y 482.467,Z 983.638,A -85,B 0,C 180,E1 -12485.904,E2 -12485.904} C_VEL
LIN {X 0,Y 479.877,Z 995.452,A -85,B 0,C 180,E1 -12488.101,E2 -12488.101} C_VEL
LIN {X 0,Y 477.214,Z 1008.531,A -85,B 0,C 180,E1 -12490.922,E2 -12490.922} C_VEL
LIN {X 0,Y 475.439,Z 1018.17,A -85,B 0,C 180,E1 -12493.38,E2 -12493.38} C_VEL
LIN {X 0,Y 473.969,Z 1027.637,A -85,B 0,C 180,E1 -12496.209,E2 -12496.209} C_VEL
LIN {X 0,Y 472.98,Z 1035.212,A -85,B 0,C 180,E1 -12499.032,E2 -12499.032} C_VEL
LIN {X 0,Y 472.403,Z 1041.087,A -85,B 0,C 180,E1 -12501.725,E2 -12501.725} C_VEL
LIN {X 0,Y 472.095,Z 1045.818,A -85,B 0,C 180,E1 -12504.653,E2 -12504.653} C_VEL
LIN {X 0,Y 471.981,Z 1048.666,A -85,B 0,C 180,E1 -12507.207,E2 -12507.207} C_VEL
LIN {X 0,Y 471.951,Z 1050.529,A -85,B 0,C 180,E1 -12510.036,E2 -12510.036} C_VEL
LIN {X 0,Y 471.933,Z 1050.767,A -85,B 0,C 180,E1 -12512.915,E2 -12512.915} C_VEL
LIN {X 0,Y 471.954,Z 1049.871,A -85,B 0,C 180,E1 -12515.349,E2 -12515.349} C_VEL
LIN {X 0,Y 472.044,Z 1047.586,A -85,B 0,C 180,E1 -12518.159,E2 -12518.159} C_VEL
LIN {X 0,Y 472.23,Z 1043.669,A -85,B 0,C 180,E1 -12520.986,E2 -12520.986} C_VEL
LIN {X 0,Y 472.641,Z 1038.856,A -85,B 0,C 180,E1 -12523.581,E2 -12523.581} C_VEL
LIN {X 0,Y 473.523,Z 1031.375,A -85,B 0,C 180,E1 -12526.689,E2 -12526.689} C_VEL
LIN {X 0,Y 474.623,Z 1023.93,A -85,B 0,C 180,E1 -12529.187,E2 -12529.187} C_VEL
LIN {X 0,Y 476.439,Z 1013.732,A -85,B 0,C 180,E1 -12532.065,E2 -12532.065} C_VEL
LIN {X 0,Y 478.686,Z 1002.549,A -85,B 0,C 180,E1 -12534.694,E2 -12534.694} C_VEL
LIN {X 0,Y 481.571,Z 989.664,A -85,B 0,C 180,E1 -12537.314,E2 -12537.314} C_VEL
LIN {X 0,Y 484.842,Z 975.551,A -85,B 0,C 180,E1 -12539.746,E2 -12539.746} C_VEL
LIN {X 0,Y 488.67,Z 959.912,A -85,B 0,C 180,E1 -12542.101,E2 -12542.101} C_VEL
LIN {X 0,Y 492.747,Z 942.996,A -85,B 0,C 180,E1 -12544.271,E2 -12544.271} C_VEL
LIN {X 0,Y 497.039,Z 925.273,A -85,B 0,C 180,E1 -12546.259,E2 -12546.259} C_VEL
LIN {X 0,Y 501.465,Z 905.971,A -85,B 0,C 180,E1 -12548.103,E2 -12548.103} C_VEL
LIN {X 0,Y 505.714,Z 886.807,A -85,B 0,C 180,E1 -12549.69,E2 -12549.69} C_VEL
LIN {X 0,Y 510.061,Z 865.297,A -85,B 0,C 180,E1 -12551.199,E2 -12551.199} C_VEL
LIN {X 0,Y 513.423,Z 847.177,A -85,B 0,C 180,E1 -12552.288,E2 -12552.288} C_VEL
LIN {X 0,Y 517.343,Z 823.726,A -85,B 0,C 180,E1 -12553.476,E2 -12553.476} C_VEL
LIN {X 0,Y 520.212,Z 803.366,A -85,B 0,C 180,E1 -12554.321,E2 -12554.321} C_VEL
LIN {X 0,Y 522.826,Z 781.873,A -85,B 0,C 180,E1 -12555.051,E2 -12555.051} C_VEL
LIN {X 0,Y 525.117,Z 757.355,A -85,B 0,C 180,E1 -12555.684,E2 -12555.684} C_VEL
LIN {X 0,Y 526.51,Z 735.76,A -85,B 0,C 180,E1 -12556.093,E2 -12556.093} C_VEL
LIN {X 0,Y 536.423,Z 486.99,A -85,B 0,C 180,E1 -12559.793,E2 -12559.793} C_VEL
LIN {X 0,Y 537.887,Z 449.193,A -85,B 0,C 180,E1 -12560.369,E2 -12560.369} C_VEL
LIN {X 0,Y 526.627,Z 430.909,A -85,B 0,C 180,E1 -12562.208,E2 -12562.208} C_VEL
LIN {X 0,Y 515.323,Z 415.027,A -85,B 0,C 180,E1 -12564.162,E2 -12564.162} C_VEL
LIN {X 0,Y 505.137,Z 401.359,A -85,B 0,C 180,E1 -12566.068,E2 -12566.068} C_VEL
LIN {X 0,Y 497.21,Z 391.268,A -85,B 0,C 180,E1 -12567.661,E2 -12567.661} C_VEL
LIN {X 0,Y 492.535,Z 385.487,A -85,B 0,C 180,E1 -12568.653,E2 -12568.653} C_VEL
LIN {X 0,Y 489.056,Z 380.901,A -85,B 0,C 180,E1 -12569.431,E2 -12569.431} C_VEL
LIN {X 0,Y 485.457,Z 377.109,A -85,B 0,C 180,E1 -12570.239,E2 -12570.239} C_VEL
LIN {X 0,Y 483.938,Z 374.706,A -85,B 0,C 180,E1 -12570.612,E2 -12570.612} C_VEL
LIN {X 0,Y 480.759,Z 371.783,A -85,B 0,C 180,E1 -12571.354,E2 -12571.354} C_VEL
LIN {X 0,Y 478.908,Z 368.519,A -85,B 0,C 180,E1 -12571.845,E2 -12571.845} C_VEL
LIN {X 0,Y 475.901,Z 366.357,A -85,B 0,C 180,E1 -12572.57,E2 -12572.57} C_VEL
LIN {X 0,Y 474.353,Z 363.538,A -85,B 0,C 180,E1 -12573.008,E2 -12573.008} C_VEL
LIN {X 0,Y 474.067,Z 362.181,A -85,B 0,C 180,E1 -12573.148,E2 -12573.148} C_VEL
LIN {X 0,Y 474.061,Z 362.181,A -85,B 0,C 180,E1 -12576.77,E2 -12576.77} C_VEL
LIN {X 0,Y 474.095,Z 362.177,A -85,B 0,C 180,E1 -12580.278,E2 -12580.278} C_VEL
LIN {X 0,Y 474.101,Z 362.174,A -85,B 0,C 180,E1 -12583.836,E2 -12583.836} C_VEL
LIN {X 0,Y 474.06,Z 362.171,A -85,B 0,C 180,E1 -12587.329,E2 -12587.329} C_VEL
LIN {X 0,Y 474.056,Z 362.163,A -85,B 0,C 180,E1 -12591.02,E2 -12591.02} C_VEL
LIN {X 0,Y 474.095,Z 362.151,A -85,B 0,C 180,E1 -12594.433,E2 -12594.433} C_VEL
LIN {X 0,Y 474.085,Z 362.155,A -85,B 0,C 180,E1 -12597.945,E2 -12597.945} C_VEL
LIN {X 0,Y 474.057,Z 362.173,A -85,B 0,C 180,E1 -12601.45,E2 -12601.45} C_VEL
LIN {X 0,Y 474.063,Z 362.18,A -85,B 0,C 180,E1 -12605.082,E2 -12605.082} C_VEL
LIN {X 0,Y 474.103,Z 362.165,A -85,B 0,C 180,E1 -12608.612,E2 -12608.612} C_VEL
LIN {X 0,Y 474.084,Z 362.154,A -85,B 0,C 180,E1 -12612.176,E2 -12612.176} C_VEL
LIN {X 0,Y 474.053,Z 362.153,A -85,B 0,C 180,E1 -12615.663,E2 -12615.663} C_VEL
LIN {X 0,Y 474.065,Z 362.152,A -85,B 0,C 180,E1 -12619.21,E2 -12619.21} C_VEL
LIN {X 0,Y 474.119,Z 362.15,A -85,B 0,C 180,E1 -12622.702,E2 -12622.702} C_VEL
LIN {X 0,Y 474.078,Z 362.158,A -85,B 0,C 180,E1 -12626.314,E2 -12626.314} C_VEL
LIN {X 0,Y 474.077,Z 362.315,A -85,B 0,C 180,E1 -12627.646,E2 -12627.646} C_VEL
LIN {X 0,Y 475.302,Z 365.501,A -85,B 0,C 180,E1 -12628.525,E2 -12628.525} C_VEL
LIN {X 0,Y 476.519,Z 367.356,A -85,B 0,C 180,E1 -12629.131,E2 -12629.131} C_VEL
LIN {X 0,Y 477.305,Z 369.143,A -85,B 0,C 180,E1 -12629.492,E2 -12629.492} C_VEL
LIN {X 0,Y 481.628,Z 374.484,A -85,B 0,C 180,E1 -12630.573,E2 -12630.573} C_VEL
LIN {X 0,Y 485.846,Z 379.99,A -85,B 0,C 180,E1 -12631.586,E2 -12631.586} C_VEL
LIN {X 0,Y 489.056,Z 383.993,A -85,B 0,C 180,E1 -12632.32,E2 -12632.32} C_VEL
LIN {X 0,Y 496.592,Z 394.098,A -85,B 0,C 180,E1 -12633.969,E2 -12633.969} C_VEL
LIN {X 0,Y 508.11,Z 410.227,A -85,B 0,C 180,E1 -12636.288,E2 -12636.288} C_VEL
LIN {X 0,Y 520.51,Z 429.063,A -85,B 0,C 180,E1 -12638.571,E2 -12638.571} C_VEL
LIN {X 0,Y 532.363,Z 448.497,A -85,B 0,C 180,E1 -12640.584,E2 -12640.584} C_VEL
LIN {X 0,Y 537.829,Z 458.36,A -85,B 0,C 180,E1 -12641.474,E2 -12641.474} C_VEL
LIN {X 0,Y 527.95,Z 707.107,A -85,B 0,C 180,E1 -12645.17,E2 -12645.17} C_VEL
LIN {X 0,Y 525.528,Z 765.296,A -85,B 0,C 180,E1 -12646.058,E2 -12646.058} C_VEL
LIN {X 0,Y 523.396,Z 790.049,A -85,B 0,C 180,E1 -12646.596,E2 -12646.596} C_VEL
LIN {X 0,Y 521.086,Z 810.719,A -85,B 0,C 180,E1 -12647.187,E2 -12647.187} C_VEL
LIN {X 0,Y 517.774,Z 835.01,A -85,B 0,C 180,E1 -12648.074,E2 -12648.074} C_VEL
LIN {X 0,Y 514.5,Z 855.632,A -85,B 0,C 180,E1 -12649.012,E2 -12649.012} C_VEL
LIN {X 0,Y 510.642,Z 877.43,A -85,B 0,C 180,E1 -12650.186,E2 -12650.186} C_VEL
LIN {X 0,Y 506.471,Z 898.347,A -85,B 0,C 180,E1 -12651.546,E2 -12651.546} C_VEL
LIN {X 0,Y 502.284,Z 918.212,A -85,B 0,C 180,E1 -12653.045,E2 -12653.045} C_VEL
LIN {X 0,Y 497.705,Z 938.553,A -85,B 0,C 180,E1 -12654.852,E2 -12654.852} C_VEL
LIN {X 0,Y 493.798,Z 955.453,A -85,B 0,C 180,E1 -12656.58,E2 -12656.58} C_VEL
LIN {X 0,Y 489.242,Z 974.735,A -85,B 0,C 180,E1 -12658.864,E2 -12658.864} C_VEL
LIN {X 0,Y 485.715,Z 989.848,A -85,B 0,C 180,E1 -12660.933,E2 -12660.933} C_VEL
LIN {X 0,Y 482.023,Z 1006.171,A -85,B 0,C 180,E1 -12663.513,E2 -12663.513} C_VEL
LIN {X 0,Y 479.406,Z 1018.351,A -85,B 0,C 180,E1 -12665.74,E2 -12665.74} C_VEL
LIN {X 0,Y 476.858,Z 1031.376,A -85,B 0,C 180,E1 -12668.473,E2 -12668.473} C_VEL
LIN {X 0,Y 475.034,Z 1041.882,A -85,B 0,C 180,E1 -12671.086,E2 -12671.086} C_VEL
LIN {X 0,Y 473.667,Z 1051.389,A -85,B 0,C 180,E1 -12673.84,E2 -12673.84} C_VEL
LIN {X 0,Y 472.751,Z 1059.313,A -85,B 0,C 180,E1 -12676.671,E2 -12676.671} C_VEL
LIN {X 0,Y 472.269,Z 1065.163,A -85,B 0,C 180,E1 -12679.231,E2 -12679.231} C_VEL
LIN {X 0,Y 471.994,Z 1070.392,A -85,B 0,C 180,E1 -12682.208,E2 -12682.208} C_VEL
LIN {X 0,Y 471.942,Z 1073.478,A -85,B 0,C 180,E1 -12684.773,E2 -12684.773} C_VEL
LIN {X 0,Y 471.932,Z 1075.375,A -85,B 0,C 180,E1 -12687.328,E2 -12687.328} C_VEL
LIN {X 0,Y 471.932,Z 1076.059,A -85,B 0,C 180,E1 -12690.243,E2 -12690.243} C_VEL
LIN {X 0,Y 471.934,Z 1075.268,A -85,B 0,C 180,E1 -12692.793,E2 -12692.793} C_VEL
LIN {X 0,Y 471.944,Z 1073.375,A -85,B 0,C 180,E1 -12695.267,E2 -12695.267} C_VEL
LIN {X 0,Y 472.022,Z 1069.754,A -85,B 0,C 180,E1 -12698.159,E2 -12698.159} C_VEL
LIN {X 0,Y 472.281,Z 1064.788,A -85,B 0,C 180,E1 -12700.861,E2 -12700.861} C_VEL
LIN {X 0,Y 472.774,Z 1058.76,A -85,B 0,C 180,E1 -12703.453,E2 -12703.453} C_VEL
LIN {X 0,Y 473.804,Z 1049.706,A -85,B 0,C 180,E1 -12706.553,E2 -12706.553} C_VEL
LIN {X 0,Y 475.071,Z 1040.927,A -85,B 0,C 180,E1 -12709.04,E2 -12709.04} C_VEL
LIN {X 0,Y 477.104,Z 1029.013,A -85,B 0,C 180,E1 -12711.903,E2 -12711.903} C_VEL
LIN {X 0,Y 479.435,Z 1016.819,A -85,B 0,C 180,E1 -12714.39,E2 -12714.39} C_VEL
LIN {X 0,Y 482.539,Z 1002.044,A -85,B 0,C 180,E1 -12716.997,E2 -12716.997} C_VEL
LIN {X 0,Y 485.708,Z 987.476,A -85,B 0,C 180,E1 -12719.207,E2 -12719.207} C_VEL
LIN {X 0,Y 489.566,Z 970.579,A -85,B 0,C 180,E1 -12721.455,E2 -12721.455} C_VEL
LIN {X 0,Y 493.463,Z 953.107,A -85,B 0,C 180,E1 -12723.446,E2 -12723.446} C_VEL
LIN {X 0,Y 497.58,Z 934.629,A -85,B 0,C 180,E1 -12725.291,E2 -12725.291} C_VEL
LIN {X 0,Y 501.813,Z 914.624,A -85,B 0,C 180,E1 -12726.995,E2 -12726.995} C_VEL
LIN {X 0,Y 505.617,Z 895.798,A -85,B 0,C 180,E1 -12728.386,E2 -12728.386} C_VEL
LIN {X 0,Y 509.903,Z 872.784,A -85,B 0,C 180,E1 -12729.827,E2 -12729.827} C_VEL
LIN {X 0,Y 513.29,Z 852.643,A -85,B 0,C 180,E1 -12730.884,E2 -12730.884} C_VEL
LIN {X 0,Y 516.792,Z 829.09,A -85,B 0,C 180,E1 -12731.912,E2 -12731.912} C_VEL
LIN {X 0,Y 519.471,Z 807.679,A -85,B 0,C 180,E1 -12732.656,E2 -12732.656} C_VEL
LIN {X 0,Y 521.774,Z 785.823,A -85,B 0,C 180,E1 -12733.26,E2 -12733.26} C_VEL
LIN {X 0,Y 523.623,Z 760.497,A -85,B 0,C 180,E1 -12733.77,E2 -12733.77} C_VEL
LIN {X 0,Y 532.185,Z 531.136,A -85,B 0,C 180,E1 -12737.175,E2 -12737.175} C_VEL
LIN {X 0,Y 534.969,Z 456.72,A -85,B 0,C 180,E1 -12738.288,E2 -12738.288} C_VEL
LIN {X 0,Y 522.845,Z 435.554,A -85,B 0,C 180,E1 -12740.177,E2 -12740.177} C_VEL
LIN {X 0,Y 511.086,Z 416.727,A -85,B 0,C 180,E1 -12742.133,E2 -12742.133} C_VEL
LIN {X 0,Y 500.477,Z 400.882,A -85,B 0,C 180,E1 -12744.029,E2 -12744.029} C_VEL
LIN {X 0,Y 490.284,Z 386.534,A -85,B 0,C 180,E1 -12745.992,E2 -12745.992} C_VEL
LIN {X 0,Y 486.274,Z 381.192,A -85,B 0,C 180,E1 -12746.806,E2 -12746.806} C_VEL
LIN {X 0,Y 481.995,Z 375.418,A -85,B 0,C 180,E1 -12747.712,E2 -12747.712} C_VEL
LIN {X 0,Y 476.729,Z 368.369,A -85,B 0,C 180,E1 -12748.938,E2 -12748.938} C_VEL
LIN {X 0,Y 475.888,Z 366.287,A -85,B 0,C 180,E1 -12749.438,E2 -12749.438} C_VEL
LIN {X 0,Y 474.21,Z 363.024,A -85,B 0,C 180,E1 -12750.31,E2 -12750.31} C_VEL
LIN {X 0,Y 474.064,Z 362.171,A -85,B 0,C 180,E1 -12750.495,E2 -12750.495} C_VEL
LIN {X 0,Y 474.057,Z 362.168,A -85,B 0,C 180,E1 -12754.112,E2 -12754.112} C_VEL
LIN {X 0,Y 474.081,Z 362.155,A -85,B 0,C 180,E1 -12757.688,E2 -12757.688} C_VEL
LIN {X 0,Y 474.102,Z 362.144,A -85,B 0,C 180,E1 -12761.253,E2 -12761.253} C_VEL
LIN {X 0,Y 474.061,Z 362.157,A -85,B 0,C 180,E1 -12764.713,E2 -12764.713} C_VEL
LIN {X 0,Y 474.06,Z 362.179,A -85,B 0,C 180,E1 -12768.318,E2 -12768.318} C_VEL
LIN {X 0,Y 474.087,Z 362.157,A -85,B 0,C 180,E1 -12771.876,E2 -12771.876} C_VEL
LIN {X 0,Y 474.083,Z 362.143,A -85,B 0,C 180,E1 -12775.282,E2 -12775.282} C_VEL
LIN {X 0,Y 474.058,Z 362.177,A -85,B 0,C 180,E1 -12778.791,E2 -12778.791} C_VEL
LIN {X 0,Y 474.062,Z 362.164,A -85,B 0,C 180,E1 -12782.418,E2 -12782.418} C_VEL
LIN {X 0,Y 474.104,Z 362.14,A -85,B 0,C 180,E1 -12785.932,E2 -12785.932} C_VEL
LIN {X 0,Y 474.074,Z 362.171,A -85,B 0,C 180,E1 -12789.347,E2 -12789.347} C_VEL
LIN {X 0,Y 474.059,Z 362.17,A -85,B 0,C 180,E1 -12792.919,E2 -12792.919} C_VEL
LIN {X 0,Y 474.078,Z 362.146,A -85,B 0,C 180,E1 -12796.417,E2 -12796.417} C_VEL
LIN {X 0,Y 474.111,Z 362.15,A -85,B 0,C 180,E1 -12799.978,E2 -12799.978} C_VEL
LIN {X 0,Y 474.072,Z 362.179,A -85,B 0,C 180,E1 -12803.493,E2 -12803.493} C_VEL
LIN {X 0,Y 474.063,Z 362.176,A -85,B 0,C 180,E1 -12807.117,E2 -12807.117} C_VEL
LIN {X 0,Y 474.078,Z 362.162,A -85,B 0,C 180,E1 -12810.691,E2 -12810.691} C_VEL
LIN {X 0,Y 474.091,Z 362.308,A -85,B 0,C 180,E1 -12812.858,E2 -12812.858} C_VEL
LIN {X 0,Y 475.104,Z 365.228,A -85,B 0,C 180,E1 -12813.139,E2 -12813.139} C_VEL
LIN {X 0,Y 477.626,Z 367.858,A -85,B 0,C 180,E1 -12813.695,E2 -12813.695} C_VEL
LIN {X 0,Y 478.935,Z 368.872,A -85,B 0,C 180,E1 -12813.968,E2 -12813.968} C_VEL
LIN {X 0,Y 481.212,Z 372.548,A -85,B 0,C 180,E1 -12814.487,E2 -12814.487} C_VEL
LIN {X 0,Y 483.785,Z 375.045,A -85,B 0,C 180,E1 -12815.016,E2 -12815.016} C_VEL
LIN {X 0,Y 486.936,Z 379.219,A -85,B 0,C 180,E1 -12815.674,E2 -12815.674} C_VEL
LIN {X 0,Y 488.583,Z 381.187,A -85,B 0,C 180,E1 -12816.006,E2 -12816.006} C_VEL
LIN {X 0,Y 492.304,Z 385.682,A -85,B 0,C 180,E1 -12816.737,E2 -12816.737} C_VEL
LIN {X 0,Y 504.843,Z 402.265,A -85,B 0,C 180,E1 -12819.071,E2 -12819.071} C_VEL
LIN {X 0,Y 517.409,Z 419.65,A -85,B 0,C 180,E1 -12821.204,E2 -12821.204} C_VEL
LIN {X 0,Y 527.401,Z 434.855,A -85,B 0,C 180,E1 -12822.794,E2 -12822.794} C_VEL
LIN {X 0,Y 535.203,Z 448.272,A -85,B 0,C 180,E1 -12823.993,E2 -12823.993} C_VEL
LIN {X 0,Y 525.815,Z 696.321,A -85,B 0,C 180,E1 -12827.658,E2 -12827.658} C_VEL
LIN {X 0,Y 523.772,Z 746.313,A -85,B 0,C 180,E1 -12828.425,E2 -12828.425} C_VEL
LIN {X 0,Y 521.832,Z 770.517,A -85,B 0,C 180,E1 -12828.974,E2 -12828.974} C_VEL
LIN {X 0,Y 519.46,Z 793.618,A -85,B 0,C 180,E1 -12829.665,E2 -12829.665} C_VEL
LIN {X 0,Y 516.413,Z 817.049,A -85,B 0,C 180,E1 -12830.574,E2 -12830.574} C_VEL
LIN {X 0,Y 513.235,Z 838.261,A -85,B 0,C 180,E1 -12831.576,E2 -12831.576} C_VEL
LIN {X 0,Y 509.311,Z 860.899,A -85,B 0,C 180,E1 -12832.865,E2 -12832.865} C_VEL
LIN {X 0,Y 505.778,Z 879.483,A -85,B 0,C 180,E1 -12834.115,E2 -12834.115} C_VEL
LIN {X 0,Y 501.402,Z 900.777,A -85,B 0,C 180,E1 -12835.781,E2 -12835.781} C_VEL
LIN {X 0,Y 497.476,Z 918.544,A -85,B 0,C 180,E1 -12837.408,E2 -12837.408} C_VEL
LIN {X 0,Y 493.285,Z 937.085,A -85,B 0,C 180,E1 -12839.35,E2 -12839.35} C_VEL
LIN {X 0,Y 489.304,Z 954.023,A -85,B 0,C 180,E1 -12841.434,E2 -12841.434} C_VEL
LIN {X 0,Y 485.877,Z 968.772,A -85,B 0,C 180,E1 -12843.495,E2 -12843.495} C_VEL
LIN {X 0,Y 483.874,Z 973.63,A -85,B 0,C 180,E1 -12844.171,E2 -12844.171} C_VEL
LIN {X 0,Y 475.222,Z 986.194,A -85,B 0,C 180,E1 -12845.939,E2 -12845.939} C_VEL
LIN {X 0,Y 473.68,Z 989.946,A -85,B 0,C 180,E1 -12846.576,E2 -12846.576} C_VEL
LIN {X 0,Y 470.77,Z 1002.847,A -85,B 0,C 180,E1 -12849.225,E2 -12849.225} C_VEL
LIN {X 0,Y 468.526,Z 1013.891,A -85,B 0,C 180,E1 -12851.845,E2 -12851.845} C_VEL
LIN {X 0,Y 466.697,Z 1023.986,A -85,B 0,C 180,E1 -12854.721,E2 -12854.721} C_VEL
LIN {X 0,Y 465.534,Z 1031.723,A -85,B 0,C 180,E1 -12857.345,E2 -12857.345} C_VEL
LIN {X 0,Y 464.646,Z 1039.108,A -85,B 0,C 180,E1 -12860.462,E2 -12860.462} C_VEL
LIN {X 0,Y 464.235,Z 1043.881,A -85,B 0,C 180,E1 -12863.072,E2 -12863.072} C_VEL
LIN {X 0,Y 464.026,Z 1047.9,A -85,B 0,C 180,E1 -12866.046,E2 -12866.046} C_VEL
LIN {X 0,Y 463.956,Z 1050.135,A -85,B 0,C 180,E1 -12868.889,E2 -12868.889} C_VEL
LIN {X 0,Y 463.931,Z 1050.997,A -85,B 0,C 180,E1 -12871.359,E2 -12871.359} C_VEL
LIN {X 0,Y 463.948,Z 1050.673,A -85,B 0,C 180,E1 -12874.326,E2 -12874.326} C_VEL
LIN {X 0,Y 463.995,Z 1048.902,A -85,B 0,C 180,E1 -12877.056,E2 -12877.056} C_VEL
LIN {X 0,Y 464.117,Z 1046.206,A -85,B 0,C 180,E1 -12879.549,E2 -12879.549} C_VEL
LIN {X 0,Y 464.468,Z 1041.533,A -85,B 0,C 180,E1 -12882.558,E2 -12882.558} C_VEL
LIN {X 0,Y 465.106,Z 1035.651,A -85,B 0,C 180,E1 -12885.333,E2 -12885.333} C_VEL
LIN {X 0,Y 466.216,Z 1028.038,A -85,B 0,C 180,E1 -12888.248,E2 -12888.248} C_VEL
LIN {X 0,Y 467.861,Z 1018.5,A -85,B 0,C 180,E1 -12891.173,E2 -12891.173} C_VEL
LIN {X 0,Y 469.943,Z 1008.241,A -85,B 0,C 180,E1 -12893.845,E2 -12893.845} C_VEL
LIN {X 0,Y 472.807,Z 995.484,A -85,B 0,C 180,E1 -12896.637,E2 -12896.637} C_VEL
LIN {X 0,Y 475.941,Z 982.559,A -85,B 0,C 180,E1 -12899.077,E2 -12899.077} C_VEL
LIN {X 0,Y 479.752,Z 967.335,A -85,B 0,C 180,E1 -12901.542,E2 -12901.542} C_VEL
LIN {X 0,Y 483.558,Z 952.326,A -85,B 0,C 180,E1 -12903.653,E2 -12903.653} C_VEL
LIN {X 0,Y 488.246,Z 933.889,A -85,B 0,C 180,E1 -12905.89,E2 -12905.89} C_VEL
LIN {X 0,Y 492.302,Z 917.405,A -85,B 0,C 180,E1 -12907.617,E2 -12907.617} C_VEL
LIN {X 0,Y 496.988,Z 897.686,A -85,B 0,C 180,E1 -12909.414,E2 -12909.414} C_VEL
LIN {X 0,Y 501.299,Z 877.962,A -85,B 0,C 180,E1 -12910.94,E2 -12910.94} C_VEL
LIN {X 0,Y 505.556,Z 857.141,A -85,B 0,C 180,E1 -12912.328,E2 -12912.328} C_VEL
LIN {X 0,Y 509.508,Z 835.23,A -85,B 0,C 180,E1 -12913.537,E2 -12913.537} C_VEL
LIN {X 0,Y 512.898,Z 813.978,A -85,B 0,C 180,E1 -12914.525,E2 -12914.525} C_VEL
LIN {X 0,Y 516.16,Z 789.465,A -85,B 0,C 180,E1 -12915.435,E2 -12915.435} C_VEL
LIN {X 0,Y 518.534,Z 767.49,A -85,B 0,C 180,E1 -12916.073,E2 -12916.073} C_VEL
LIN {X 0,Y 520.571,Z 741.414,A -85,B 0,C 180,E1 -12916.623,E2 -12916.623} C_VEL
LIN {X 0,Y 530.099,Z 511.807,A -85,B 0,C 180,E1 -12920.075,E2 -12920.075} C_VEL
LIN {X 0,Y 532.528,Z 452.842,A -85,B 0,C 180,E1 -12920.971,E2 -12920.971} C_VEL
LIN {X 0,Y 522.36,Z 436.353,A -85,B 0,C 180,E1 -12922.676,E2 -12922.676} C_VEL
LIN {X 0,Y 510.049,Z 418.773,A -85,B 0,C 180,E1 -12924.874,E2 -12924.874} C_VEL
LIN {X 0,Y 498.444,Z 403.366,A -85,B 0,C 180,E1 -12927.137,E2 -12927.137} C_VEL
LIN {X 0,Y 493.337,Z 397.077,A -85,B 0,C 180,E1 -12928.199,E2 -12928.199} C_VEL
LIN {X 0,Y 489.447,Z 392.132,A -85,B 0,C 180,E1 -12929.049,E2 -12929.049} C_VEL
LIN {X 0,Y 485.415,Z 387.125,A -85,B 0,C 180,E1 -12929.964,E2 -12929.964} C_VEL
LIN {X 0,Y 481.938,Z 382.81,A -85,B 0,C 180,E1 -12930.785,E2 -12930.785} C_VEL
LIN {X 0,Y 480.711,Z 381.436,A -85,B 0,C 180,E1 -12931.079,E2 -12931.079} C_VEL
LIN {X 0,Y 477.53,Z 377.878,A -85,B 0,C 180,E1 -12931.859,E2 -12931.859} C_VEL
LIN {X 0,Y 476.191,Z 375.752,A -85,B 0,C 180,E1 -12932.215,E2 -12932.215} C_VEL
LIN {X 0,Y 473.057,Z 372.975,A -85,B 0,C 180,E1 -12933.005,E2 -12933.005} C_VEL
LIN {X 0,Y 471.22,Z 369.639,A -85,B 0,C 180,E1 -12933.538,E2 -12933.538} C_VEL
LIN {X 0,Y 467.964,Z 367.324,A -85,B 0,C 180,E1 -12934.396,E2 -12934.396} C_VEL
LIN {X 0,Y 466.4,Z 364.474,A -85,B 0,C 180,E1 -12934.882,E2 -12934.882} C_VEL
LIN {X 0,Y 466.12,Z 363.148,A -85,B 0,C 180,E1 -12935.002,E2 -12935.002} C_VEL
LIN {X 0,Y 466.127,Z 363.146,A -85,B 0,C 180,E1 -12938.613,E2 -12938.613} C_VEL
LIN {X 0,Y 466.163,Z 363.141,A -85,B 0,C 180,E1 -12942.138,E2 -12942.138} C_VEL
LIN {X 0,Y 466.146,Z 363.143,A -85,B 0,C 180,E1 -12945.719,E2 -12945.719} C_VEL
LIN {X 0,Y 466.118,Z 363.151,A -85,B 0,C 180,E1 -12949.258,E2 -12949.258} C_VEL
LIN {X 0,Y 466.121,Z 363.16,A -85,B 0,C 180,E1 -12952.977,E2 -12952.977} C_VEL
LIN {X 0,Y 466.15,Z 363.166,A -85,B 0,C 180,E1 -12956.557,E2 -12956.557} C_VEL
LIN {X 0,Y 466.178,Z 363.156,A -85,B 0,C 180,E1 -12960.246,E2 -12960.246} C_VEL
LIN {X 0,Y 466.138,Z 363.149,A -85,B 0,C 180,E1 -12963.936,E2 -12963.936} C_VEL
LIN {X 0,Y 466.114,Z 363.143,A -85,B 0,C 180,E1 -12967.519,E2 -12967.519} C_VEL
LIN {X 0,Y 466.124,Z 363.141,A -85,B 0,C 180,E1 -12971.132,E2 -12971.132} C_VEL
LIN {X 0,Y 466.17,Z 363.14,A -85,B 0,C 180,E1 -12974.681,E2 -12974.681} C_VEL
LIN {X 0,Y 466.156,Z 363.147,A -85,B 0,C 180,E1 -12978.38,E2 -12978.38} C_VEL
LIN {X 0,Y 466.12,Z 363.16,A -85,B 0,C 180,E1 -12981.917,E2 -12981.917} C_VEL
LIN {X 0,Y 466.12,Z 363.164,A -85,B 0,C 180,E1 -12985.542,E2 -12985.542} C_VEL
LIN {X 0,Y 466.144,Z 363.338,A -85,B 0,C 180,E1 -12985.95,E2 -12985.95} C_VEL
LIN {X 0,Y 467.734,Z 367.014,A -85,B 0,C 180,E1 -12987.087,E2 -12987.087} C_VEL
LIN {X 0,Y 468.874,Z 368.515,A -85,B 0,C 180,E1 -12987.531,E2 -12987.531} C_VEL
LIN {X 0,Y 471.856,Z 372.619,A -85,B 0,C 180,E1 -12988.372,E2 -12988.372} C_VEL
LIN {X 0,Y 474.05,Z 375.053,A -85,B 0,C 180,E1 -12988.952,E2 -12988.952} C_VEL
LIN {X 0,Y 477.533,Z 379.466,A -85,B 0,C 180,E1 -12989.856,E2 -12989.856} C_VEL
LIN {X 0,Y 486.363,Z 391.096,A -85,B 0,C 180,E1 -12991.999,E2 -12991.999} C_VEL
LIN {X 0,Y 493.35,Z 400.497,A -85,B 0,C 180,E1 -12993.559,E2 -12993.559} C_VEL
LIN {X 0,Y 504.851,Z 416.811,A -85,B 0,C 180,E1 -12995.926,E2 -12995.926} C_VEL
LIN {X 0,Y 517.021,Z 435.55,A -85,B 0,C 180,E1 -12998.216,E2 -12998.216} C_VEL
LIN {X 0,Y 528.515,Z 454.634,A -85,B 0,C 180,E1 -13000.211,E2 -13000.211} C_VEL
LIN {X 0,Y 532.466,Z 461.98,A -85,B 0,C 180,E1 -13000.875,E2 -13000.875} C_VEL
LIN {X 0,Y 522.243,Z 710.056,A -85,B 0,C 180,E1 -13004.586,E2 -13004.586} C_VEL
LIN {X 0,Y 519.837,Z 765.471,A -85,B 0,C 180,E1 -13005.441,E2 -13005.441} C_VEL
LIN {X 0,Y 517.64,Z 790.07,A -85,B 0,C 180,E1 -13005.98,E2 -13005.98} C_VEL
LIN {X 0,Y 515.264,Z 810.646,A -85,B 0,C 180,E1 -13006.572,E2 -13006.572} C_VEL
LIN {X 0,Y 511.812,Z 835.1,A -85,B 0,C 180,E1 -13007.472,E2 -13007.472} C_VEL
LIN {X 0,Y 508.624,Z 854.555,A -85,B 0,C 180,E1 -13008.359,E2 -13008.359} C_VEL
LIN {X 0,Y 504.616,Z 876.537,A -85,B 0,C 180,E1 -13009.543,E2 -13009.543} C_VEL
LIN {X 0,Y 500.294,Z 897.508,A -85,B 0,C 180,E1 -13010.909,E2 -13010.909} C_VEL
LIN {X 0,Y 496.097,Z 916.695,A -85,B 0,C 180,E1 -13012.36,E2 -13012.36} C_VEL
LIN {X 0,Y 491.136,Z 937.933,A -85,B 0,C 180,E1 -13014.247,E2 -13014.247} C_VEL
LIN {X 0,Y 487.068,Z 954.804,A -85,B 0,C 180,E1 -13015.985,E2 -13015.985} C_VEL
LIN {X 0,Y 482.433,Z 973.69,A -85,B 0,C 180,E1 -13018.235,E2 -13018.235} C_VEL
LIN {X 0,Y 478.672,Z 988.961,A -85,B 0,C 180,E1 -13020.34,E2 -13020.34} C_VEL
LIN {X 0,Y 474.792,Z 1005.322,A -85,B 0,C 180,E1 -13022.942,E2 -13022.942} C_VEL
LIN {X 0,Y 471.865,Z 1018.2,A -85,B 0,C 180,E1 -13025.327,E2 -13025.327} C_VEL
LIN {X 0,Y 469.182,Z 1031.211,A -85,B 0,C 180,E1 -13028.102,E2 -13028.102} C_VEL
LIN {X 0,Y 467.244,Z 1041.71,A -85,B 0,C 180,E1 -13030.758,E2 -13030.758} C_VEL
LIN {X 0,Y 465.744,Z 1051.561,A -85,B 0,C 180,E1 -13033.669,E2 -13033.669} C_VEL
LIN {X 0,Y 464.78,Z 1059.433,A -85,B 0,C 180,E1 -13036.565,E2 -13036.565} C_VEL
LIN {X 0,Y 464.274,Z 1065.294,A -85,B 0,C 180,E1 -13039.201,E2 -13039.201} C_VEL
LIN {X 0,Y 463.989,Z 1070.518,A -85,B 0,C 180,E1 -13042.322,E2 -13042.322} C_VEL
LIN {X 0,Y 463.943,Z 1073.39,A -85,B 0,C 180,E1 -13044.807,E2 -13044.807} C_VEL
LIN {X 0,Y 463.933,Z 1075.237,A -85,B 0,C 180,E1 -13047.406,E2 -13047.406} C_VEL
LIN {X 0,Y 463.933,Z 1075.821,A -85,B 0,C 180,E1 -13050.37,E2 -13050.37} C_VEL
LIN {X 0,Y 463.938,Z 1074.979,A -85,B 0,C 180,E1 -13052.965,E2 -13052.965} C_VEL
LIN {X 0,Y 463.945,Z 1073.072,A -85,B 0,C 180,E1 -13055.441,E2 -13055.441} C_VEL
LIN {X 0,Y 464.051,Z 1069.098,A -85,B 0,C 180,E1 -13058.55,E2 -13058.55} C_VEL
LIN {X 0,Y 464.326,Z 1064.288,A -85,B 0,C 180,E1 -13061.175,E2 -13061.175} C_VEL
LIN {X 0,Y 464.87,Z 1058.203,A -85,B 0,C 180,E1 -13063.813,E2 -13063.813} C_VEL
LIN {X 0,Y 465.933,Z 1049.446,A -85,B 0,C 180,E1 -13066.841,E2 -13066.841} C_VEL
LIN {X 0,Y 467.275,Z 1040.658,A -85,B 0,C 180,E1 -13069.37,E2 -13069.37} C_VEL
LIN {X 0,Y 469.428,Z 1028.73,A -85,B 0,C 180,E1 -13072.281,E2 -13072.281} C_VEL
LIN {X 0,Y 471.748,Z 1017.173,A -85,B 0,C 180,E1 -13074.68,E2 -13074.68} C_VEL
LIN {X 0,Y 474.803,Z 1003.351,A -85,B 0,C 180,E1 -13077.192,E2 -13077.192} C_VEL
LIN {X 0,Y 478.289,Z 987.945,A -85,B 0,C 180,E1 -13079.579,E2 -13079.579} C_VEL
LIN {X 0,Y 482.157,Z 971.697,A -85,B 0,C 180,E1 -13081.786,E2 -13081.786} C_VEL
LIN {X 0,Y 486.44,Z 953.32,A -85,B 0,C 180,E1 -13083.923,E2 -13083.923} C_VEL
LIN {X 0,Y 490.566,Z 935.499,A -85,B 0,C 180,E1 -13085.729,E2 -13085.729} C_VEL
LIN {X 0,Y 495.107,Z 914.975,A -85,B 0,C 180,E1 -13087.509,E2 -13087.509} C_VEL
LIN {X 0,Y 499.039,Z 896.208,A -85,B 0,C 180,E1 -13088.913,E2 -13088.913} C_VEL
LIN {X 0,Y 503.431,Z 873.57,A -85,B 0,C 180,E1 -13090.352,E2 -13090.352} C_VEL
LIN {X 0,Y 506.962,Z 853.296,A -85,B 0,C 180,E1 -13091.431,E2 -13091.431} C_VEL
LIN {X 0,Y 510.531,Z 830.394,A -85,B 0,C 180,E1 -13092.45,E2 -13092.45} C_VEL
LIN {X 0,Y 513.436,Z 807.939,A -85,B 0,C 180,E1 -13093.241,E2 -13093.241} C_VEL
LIN {X 0,Y 515.735,Z 786.864,A -85,B 0,C 180,E1 -13093.83,E2 -13093.83} C_VEL
LIN {X 0,Y 517.743,Z 760.82,A -85,B 0,C 180,E1 -13094.366,E2 -13094.366} C_VEL
LIN {X 0,Y 526.529,Z 534.34,A -85,B 0,C 180,E1 -13097.756,E2 -13097.756} C_VEL
LIN {X 0,Y 529.359,Z 459.98,A -85,B 0,C 180,E1 -13098.884,E2 -13098.884} C_VEL
LIN {X 0,Y 517.246,Z 438.875,A -85,B 0,C 180,E1 -13100.828,E2 -13100.828} C_VEL
LIN {X 0,Y 505.333,Z 419.769,A -85,B 0,C 180,E1 -13102.879,E2 -13102.879} C_VEL
LIN {X 0,Y 493.247,Z 401.767,A -85,B 0,C 180,E1 -13105.134,E2 -13105.134} C_VEL
LIN {X 0,Y 483.322,Z 388.058,A -85,B 0,C 180,E1 -13107.143,E2 -13107.143} C_VEL
LIN {X 0,Y 478.844,Z 382.015,A -85,B 0,C 180,E1 -13108.109,E2 -13108.109} C_VEL
LIN {X 0,Y 471.574,Z 372.628,A -85,B 0,C 180,E1 -13109.763,E2 -13109.763} C_VEL
LIN {X 0,Y 468.529,Z 368.452,A -85,B 0,C 180,E1 -13110.502,E2 -13110.502} C_VEL
LIN {X 0,Y 466.189,Z 363.557,A -85,B 0,C 180,E1 -13111.845,E2 -13111.845} C_VEL
LIN {X 0,Y 466.121,Z 363.144,A -85,B 0,C 180,E1 -13111.98,E2 -13111.98} C_VEL
LIN {X 0,Y 466.153,Z 363.146,A -85,B 0,C 180,E1 -13115.545,E2 -13115.545} C_VEL
LIN {X 0,Y 466.149,Z 363.166,A -85,B 0,C 180,E1 -13119.009,E2 -13119.009} C_VEL
LIN {X 0,Y 466.118,Z 363.156,A -85,B 0,C 180,E1 -13122.523,E2 -13122.523} C_VEL
LIN {X 0,Y 466.118,Z 363.139,A -85,B 0,C 180,E1 -13126.225,E2 -13126.225} C_VEL
LIN {X 0,Y 466.154,Z 363.134,A -85,B 0,C 180,E1 -13129.745,E2 -13129.745} C_VEL
LIN {X 0,Y 466.161,Z 363.165,A -85,B 0,C 180,E1 -13133.349,E2 -13133.349} C_VEL
LIN {X 0,Y 466.121,Z 363.148,A -85,B 0,C 180,E1 -13136.926,E2 -13136.926} C_VEL
LIN {X 0,Y 466.118,Z 363.132,A -85,B 0,C 180,E1 -13140.492,E2 -13140.492} C_VEL
LIN {X 0,Y 466.151,Z 363.159,A -85,B 0,C 180,E1 -13144.059,E2 -13144.059} C_VEL
LIN {X 0,Y 466.18,Z 363.151,A -85,B 0,C 180,E1 -13147.766,E2 -13147.766} C_VEL
LIN {X 0,Y 466.133,Z 363.13,A -85,B 0,C 180,E1 -13151.392,E2 -13151.392} C_VEL
LIN {X 0,Y 466.118,Z 363.15,A -85,B 0,C 180,E1 -13154.917,E2 -13154.917} C_VEL
LIN {X 0,Y 466.138,Z 363.169,A -85,B 0,C 180,E1 -13158.538,E2 -13158.538} C_VEL
LIN {X 0,Y 466.176,Z 363.143,A -85,B 0,C 180,E1 -13162.179,E2 -13162.179} C_VEL
LIN {X 0,Y 466.149,Z 363.136,A -85,B 0,C 180,E1 -13165.813,E2 -13165.813} C_VEL
LIN {X 0,Y 466.121,Z 363.141,A -85,B 0,C 180,E1 -13169.281,E2 -13169.281} C_VEL
LIN {X 0,Y 466.145,Z 363.332,A -85,B 0,C 180,E1 -13171.262,E2 -13171.262} C_VEL
LIN {X 0,Y 467.136,Z 366.173,A -85,B 0,C 180,E1 -13171.557,E2 -13171.557} C_VEL
LIN {X 0,Y 469.659,Z 368.809,A -85,B 0,C 180,E1 -13172.157,E2 -13172.157} C_VEL
LIN {X 0,Y 471.092,Z 369.9,A -85,B 0,C 180,E1 -13172.479,E2 -13172.479} C_VEL
LIN {X 0,Y 473.328,Z 373.522,A -85,B 0,C 180,E1 -13173.026,E2 -13173.026} C_VEL
LIN {X 0,Y 476.108,Z 376.165,A -85,B 0,C 180,E1 -13173.636,E2 -13173.636} C_VEL
LIN {X 0,Y 479.193,Z 380.342,A -85,B 0,C 180,E1 -13174.327,E2 -13174.327} C_VEL
LIN {X 0,Y 481.043,Z 382.367,A -85,B 0,C 180,E1 -13174.718,E2 -13174.718} C_VEL
LIN {X 0,Y 485.99,Z 388.713,A -85,B 0,C 180,E1 -13175.755,E2 -13175.755} C_VEL
LIN {X 0,Y 490.95,Z 395.022,A -85,B 0,C 180,E1 -13176.746,E2 -13176.746} C_VEL
LIN {X 0,Y 501.016,Z 408.196,A -85,B 0,C 180,E1 -13178.639,E2 -13178.639} C_VEL
LIN {X 0,Y 513.708,Z 425.991,A -85,B 0,C 180,E1 -13180.844,E2 -13180.844} C_VEL
LIN {X 0,Y 523.344,Z 440.79,A -85,B 0,C 180,E1 -13182.411,E2 -13182.411} C_VEL
LIN {X 0,Y 529.658,Z 451.856,A -85,B 0,C 180,E1 -13183.409,E2 -13183.409} C_VEL
LIN {X 0,Y 519.859,Z 701.39,A -85,B 0,C 180,E1 -13187.123,E2 -13187.123} C_VEL
LIN {X 0,Y 517.888,Z 747.099,A -85,B 0,C 180,E1 -13187.834,E2 -13187.834} C_VEL
LIN {X 0,Y 515.883,Z 771.168,A -85,B 0,C 180,E1 -13188.388,E2 -13188.388} C_VEL
LIN {X 0,Y 513.349,Z 795.051,A -85,B 0,C 180,E1 -13189.112,E2 -13189.112} C_VEL
LIN {X 0,Y 510.224,Z 818.004,A -85,B 0,C 180,E1 -13190.018,E2 -13190.018} C_VEL
LIN {X 0,Y 506.989,Z 838.853,A -85,B 0,C 180,E1 -13191.014,E2 -13191.014} C_VEL
LIN {X 0,Y 502.974,Z 861.197,A -85,B 0,C 180,E1 -13192.299,E2 -13192.299} C_VEL
LIN {X 0,Y 499.279,Z 879.973,A -85,B 0,C 180,E1 -13193.574,E2 -13193.574} C_VEL
LIN {X 0,Y 494.747,Z 901.22,A -85,B 0,C 180,E1 -13195.255,E2 -13195.255} C_VEL
LIN {X 0,Y 490.679,Z 918.969,A -85,B 0,C 180,E1 -13196.899,E2 -13196.899} C_VEL
LIN {X 0,Y 486.319,Z 937.478,A -85,B 0,C 180,E1 -13198.863,E2 -13198.863} C_VEL
LIN {X 0,Y 482.171,Z 954.403,A -85,B 0,C 180,E1 -13200.971,E2 -13200.971} C_VEL
LIN {X 0,Y 478.249,Z 970.673,A -85,B 0,C 180,E1 -13203.288,E2 -13203.288} C_VEL
LIN {X 0,Y 474.711,Z 985.357,A -85,B 0,C 180,E1 -13205.749,E2 -13205.749} C_VEL
LIN {X 0,Y 473.68,Z 989.946,A -85,B 0,C 180,E1 -13206.576,E2 -13206.576} C_VEL
LIN {X 0,Y 471.804,Z 994.228,A -85,B 0,C 180,E1 -13207.328,E2 -13207.328} C_VEL
LIN {X 0,Y 463.475,Z 1005.134,A -85,B 0,C 180,E1 -13209.318,E2 -13209.318} C_VEL
LIN {X 0,Y 462.054,Z 1008.223,A -85,B 0,C 180,E1 -13210.027,E2 -13210.027} C_VEL
LIN {X 0,Y 459.978,Z 1018.321,A -85,B 0,C 180,E1 -13212.674,E2 -13212.674} C_VEL
LIN {X 0,Y 458.303,Z 1027.843,A -85,B 0,C 180,E1 -13215.598,E2 -13215.598} C_VEL
LIN {X 0,Y 457.168,Z 1035.458,A -85,B 0,C 180,E1 -13218.52,E2 -13218.52} C_VEL
LIN {X 0,Y 456.528,Z 1041.112,A -85,B 0,C 180,E1 -13221.181,E2 -13221.181} C_VEL
LIN {X 0,Y 456.122,Z 1046.237,A -85,B 0,C 180,E1 -13224.41,E2 -13224.41} C_VEL
LIN {X 0,Y 455.993,Z 1049.024,A -85,B 0,C 180,E1 -13226.983,E2 -13226.983} C_VEL
LIN {X 0,Y 455.957,Z 1050.829,A -85,B 0,C 180,E1 -13229.749,E2 -13229.749} C_VEL
LIN {X 0,Y 455.936,Z 1051.23,A -85,B 0,C 180,E1 -13232.765,E2 -13232.765} C_VEL
LIN {X 0,Y 455.961,Z 1050.407,A -85,B 0,C 180,E1 -13235.285,E2 -13235.285} C_VEL
LIN {X 0,Y 456.03,Z 1048.428,A -85,B 0,C 180,E1 -13237.94,E2 -13237.94} C_VEL
LIN {X 0,Y 456.268,Z 1044.431,A -85,B 0,C 180,E1 -13241.119,E2 -13241.119} C_VEL
LIN {X 0,Y 456.698,Z 1039.948,A -85,B 0,C 180,E1 -13243.677,E2 -13243.677} C_VEL
LIN {X 0,Y 457.565,Z 1033.418,A -85,B 0,C 180,E1 -13246.635,E2 -13246.635} C_VEL
LIN {X 0,Y 458.928,Z 1025.023,A -85,B 0,C 180,E1 -13249.605,E2 -13249.605} C_VEL
LIN {X 0,Y 460.826,Z 1015.455,A -85,B 0,C 180,E1 -13252.45,E2 -13252.45} C_VEL
LIN {X 0,Y 463.387,Z 1003.91,A -85,B 0,C 180,E1 -13255.295,E2 -13255.295} C_VEL
LIN {X 0,Y 466.368,Z 991.804,A -85,B 0,C 180,E1 -13257.865,E2 -13257.865} C_VEL
LIN {X 0,Y 470.149,Z 977.028,A -85,B 0,C 180,E1 -13260.533,E2 -13260.533} C_VEL
LIN {X 0,Y 473.82,Z 963.193,A -85,B 0,C 180,E1 -13262.699,E2 -13262.699} C_VEL
LIN {X 0,Y 478.625,Z 945.105,A -85,B 0,C 180,E1 -13265.138,E2 -13265.138} C_VEL
LIN {X 0,Y 482.842,Z 928.989,A -85,B 0,C 180,E1 -13267.012,E2 -13267.012} C_VEL
LIN {X 0,Y 487.97,Z 908.659,A -85,B 0,C 180,E1 -13269.049,E2 -13269.049} C_VEL
LIN {X 0,Y 492.318,Z 890.419,A -85,B 0,C 180,E1 -13270.612,E2 -13270.612} C_VEL
LIN {X 0,Y 497.275,Z 868.075,A -85,B 0,C 180,E1 -13272.246,E2 -13272.246} C_VEL
LIN {X 0,Y 501.059,Z 849.129,A -85,B 0,C 180,E1 -13273.416,E2 -13273.416} C_VEL
LIN {X 0,Y 505.057,Z 827.238,A -85,B 0,C 180,E1 -13274.566,E2 -13274.566} C_VEL
LIN {X 0,Y 508.423,Z 805.036,A -85,B 0,C 180,E1 -13275.512,E2 -13275.512} C_VEL
LIN {X 0,Y 511.082,Z 784.633,A -85,B 0,C 180,E1 -13276.223,E2 -13276.223} C_VEL
LIN {X 0,Y 513.702,Z 759.186,A -85,B 0,C 180,E1 -13276.905,E2 -13276.905} C_VEL
LIN {X 0,Y 515.224,Z 737.466,A -85,B 0,C 180,E1 -13277.328,E2 -13277.328} C_VEL
LIN {X 0,Y 525.825,Z 490.776,A -85,B 0,C 180,E1 -13281.052,E2 -13281.052} C_VEL
LIN {X 0,Y 527.232,Z 456.53,A -85,B 0,C 180,E1 -13281.584,E2 -13281.584} C_VEL
LIN {X 0,Y 518.4,Z 442.163,A -85,B 0,C 180,E1 -13283.106,E2 -13283.106} C_VEL
LIN {X 0,Y 506.621,Z 425.172,A -85,B 0,C 180,E1 -13285.257,E2 -13285.257} C_VEL
LIN {X 0,Y 495.272,Z 409.956,A -85,B 0,C 180,E1 -13287.519,E2 -13287.519} C_VEL
LIN {X 0,Y 486.502,Z 398.885,A -85,B 0,C 180,E1 -13289.424,E2 -13289.424} C_VEL
LIN {X 0,Y 482.516,Z 393.936,A -85,B 0,C 180,E1 -13290.347,E2 -13290.347} C_VEL
LIN {X 0,Y 478.206,Z 388.608,A -85,B 0,C 180,E1 -13291.391,E2 -13291.391} C_VEL
LIN {X 0,Y 474.75,Z 384.598,A -85,B 0,C 180,E1 -13292.26,E2 -13292.26} C_VEL
LIN {X 0,Y 473.508,Z 382.871,A -85,B 0,C 180,E1 -13292.591,E2 -13292.591} C_VEL
LIN {X 0,Y 470.244,Z 379.565,A -85,B 0,C 180,E1 -13293.445,E2 -13293.445} C_VEL
LIN {X 0,Y 468.592,Z 376.914,A -85,B 0,C 180,E1 -13293.924,E2 -13293.924} C_VEL
LIN {X 0,Y 465.331,Z 374.096,A -85,B 0,C 180,E1 -13294.82,E2 -13294.82} C_VEL
LIN {X 0,Y 463.531,Z 370.718,A -85,B 0,C 180,E1 -13295.397,E2 -13295.397} C_VEL
LIN {X 0,Y 460.185,Z 368.505,A -85,B 0,C 180,E1 -13296.367,E2 -13296.367} C_VEL
LIN {X 0,Y 458.546,Z 365.742,A -85,B 0,C 180,E1 -13296.924,E2 -13296.924} C_VEL
LIN {X 0,Y 458.182,Z 364.15,A -85,B 0,C 180,E1 -13297.104,E2 -13297.104} C_VEL
LIN {X 0,Y 458.186,Z 364.15,A -85,B 0,C 180,E1 -13300.76,E2 -13300.76} C_VEL
LIN {X 0,Y 458.219,Z 364.153,A -85,B 0,C 180,E1 -13304.301,E2 -13304.301} C_VEL
LIN {X 0,Y 458.221,Z 364.153,A -85,B 0,C 180,E1 -13307.908,E2 -13307.908} C_VEL
LIN {X 0,Y 458.186,Z 364.146,A -85,B 0,C 180,E1 -13311.466,E2 -13311.466} C_VEL
LIN {X 0,Y 458.178,Z 364.137,A -85,B 0,C 180,E1 -13315.118,E2 -13315.118} C_VEL
LIN {X 0,Y 458.197,Z 364.129,A -85,B 0,C 180,E1 -13318.75,E2 -13318.75} C_VEL
LIN {X 0,Y 458.224,Z 364.129,A -85,B 0,C 180,E1 -13322.251,E2 -13322.251} C_VEL
LIN {X 0,Y 458.194,Z 364.142,A -85,B 0,C 180,E1 -13325.887,E2 -13325.887} C_VEL
LIN {X 0,Y 458.18,Z 364.159,A -85,B 0,C 180,E1 -13329.459,E2 -13329.459} C_VEL
LIN {X 0,Y 458.191,Z 364.153,A -85,B 0,C 180,E1 -13333.118,E2 -13333.118} C_VEL
LIN {X 0,Y 458.226,Z 364.135,A -85,B 0,C 180,E1 -13336.677,E2 -13336.677} C_VEL
LIN {X 0,Y 458.205,Z 364.131,A -85,B 0,C 180,E1 -13340.302,E2 -13340.302} C_VEL
LIN {X 0,Y 458.177,Z 364.133,A -85,B 0,C 180,E1 -13343.812,E2 -13343.812} C_VEL
LIN {X 0,Y 458.216,Z 364.355,A -85,B 0,C 180,E1 -13344.083,E2 -13344.083} C_VEL
LIN {X 0,Y 459.577,Z 367.733,A -85,B 0,C 180,E1 -13345.104,E2 -13345.104} C_VEL
LIN {X 0,Y 462.088,Z 370.554,A -85,B 0,C 180,E1 -13345.885,E2 -13345.885} C_VEL
LIN {X 0,Y 465.638,Z 374.677,A -85,B 0,C 180,E1 -13346.942,E2 -13346.942} C_VEL
LIN {X 0,Y 469.986,Z 380.296,A -85,B 0,C 180,E1 -13348.184,E2 -13348.184} C_VEL
LIN {X 0,Y 472.027,Z 382.917,A -85,B 0,C 180,E1 -13348.741,E2 -13348.741} C_VEL
LIN {X 0,Y 479.259,Z 392.183,A -85,B 0,C 180,E1 -13350.602,E2 -13350.602} C_VEL
LIN {X 0,Y 484.358,Z 399.161,A -85,B 0,C 180,E1 -13351.833,E2 -13351.833} C_VEL
LIN {X 0,Y 490.134,Z 406.894,A -85,B 0,C 180,E1 -13353.143,E2 -13353.143} C_VEL
LIN {X 0,Y 501.797,Z 423.689,A -85,B 0,C 180,E1 -13355.598,E2 -13355.598} C_VEL
LIN {X 0,Y 513.715,Z 442.294,A -85,B 0,C 180,E1 -13357.886,E2 -13357.886} C_VEL
LIN {X 0,Y 525.097,Z 461.488,A -85,B 0,C 180,E1 -13359.902,E2 -13359.902} C_VEL
LIN {X 0,Y 527.168,Z 465.477,A -85,B 0,C 180,E1 -13360.261,E2 -13360.261} C_VEL
LIN {X 0,Y 516.596,Z 712.931,A -85,B 0,C 180,E1 -13363.989,E2 -13363.989} C_VEL
LIN {X 0,Y 514.201,Z 765.76,A -85,B 0,C 180,E1 -13364.812,E2 -13364.812} C_VEL
LIN {X 0,Y 511.93,Z 790.227,A -85,B 0,C 180,E1 -13365.355,E2 -13365.355} C_VEL
LIN {X 0,Y 509.45,Z 811,A -85,B 0,C 180,E1 -13365.957,E2 -13365.957} C_VEL
LIN {X 0,Y 505.908,Z 835.192,A -85,B 0,C 180,E1 -13366.855,E2 -13366.855} C_VEL
LIN {X 0,Y 502.614,Z 854.609,A -85,B 0,C 180,E1 -13367.747,E2 -13367.747} C_VEL
LIN {X 0,Y 498.359,Z 877.126,A -85,B 0,C 180,E1 -13368.973,E2 -13368.973} C_VEL
LIN {X 0,Y 493.82,Z 898.296,A -85,B 0,C 180,E1 -13370.371,E2 -13370.371} C_VEL
LIN {X 0,Y 489.154,Z 918.858,A -85,B 0,C 180,E1 -13371.953,E2 -13371.953} C_VEL
LIN {X 0,Y 484.379,Z 938.312,A -85,B 0,C 180,E1 -13373.724,E2 -13373.724} C_VEL
LIN {X 0,Y 480.121,Z 955.271,A -85,B 0,C 180,E1 -13375.496,E2 -13375.496} C_VEL
LIN {X 0,Y 475.397,Z 973.705,A -85,B 0,C 180,E1 -13377.728,E2 -13377.728} C_VEL
LIN {X 0,Y 471.522,Z 988.749,A -85,B 0,C 180,E1 -13379.83,E2 -13379.83} C_VEL
LIN {X 0,Y 467.427,Z 1005.18,A -85,B 0,C 180,E1 -13382.48,E2 -13382.48} C_VEL
LIN {X 0,Y 464.352,Z 1018.05,A -85,B 0,C 180,E1 -13384.9,E2 -13384.9} C_VEL
LIN {X 0,Y 461.523,Z 1031.047,A -85,B 0,C 180,E1 -13387.72,E2 -13387.72} C_VEL
LIN {X 0,Y 459.443,Z 1041.649,A -85,B 0,C 180,E1 -13390.449,E2 -13390.449} C_VEL
LIN {X 0,Y 457.874,Z 1051.37,A -85,B 0,C 180,E1 -13393.377,E2 -13393.377} C_VEL
LIN {X 0,Y 456.835,Z 1059.329,A -85,B 0,C 180,E1 -13396.361,E2 -13396.361} C_VEL
LIN {X 0,Y 456.284,Z 1065.362,A -85,B 0,C 180,E1 -13399.137,E2 -13399.137} C_VEL
LIN {X 0,Y 455.995,Z 1070.318,A -85,B 0,C 180,E1 -13402.186,E2 -13402.186} C_VEL
LIN {X 0,Y 455.944,Z 1073.186,A -85,B 0,C 180,E1 -13404.715,E2 -13404.715} C_VEL
LIN {X 0,Y 455.935,Z 1075.029,A -85,B 0,C 180,E1 -13407.36,E2 -13407.36} C_VEL
LIN {X 0,Y 455.936,Z 1075.605,A -85,B 0,C 180,E1 -13410.377,E2 -13410.377} C_VEL
LIN {X 0,Y 455.94,Z 1074.759,A -85,B 0,C 180,E1 -13413.017,E2 -13413.017} C_VEL
LIN {X 0,Y 455.947,Z 1072.847,A -85,B 0,C 180,E1 -13415.537,E2 -13415.537} C_VEL
LIN {X 0,Y 456.052,Z 1069.07,A -85,B 0,C 180,E1 -13418.576,E2 -13418.576} C_VEL
LIN {X 0,Y 456.354,Z 1064.045,A -85,B 0,C 180,E1 -13421.373,E2 -13421.373} C_VEL
LIN {X 0,Y 456.974,Z 1057.644,A -85,B 0,C 180,E1 -13424.186,E2 -13424.186} C_VEL
LIN {X 0,Y 458.072,Z 1049.184,A -85,B 0,C 180,E1 -13427.138,E2 -13427.138} C_VEL
LIN {X 0,Y 459.49,Z 1040.389,A -85,B 0,C 180,E1 -13429.712,E2 -13429.712} C_VEL
LIN {X 0,Y 461.815,Z 1028.187,A -85,B 0,C 180,E1 -13432.728,E2 -13432.728} C_VEL
LIN {X 0,Y 464.219,Z 1016.881,A -85,B 0,C 180,E1 -13435.108,E2 -13435.108} C_VEL
LIN {X 0,Y 467.596,Z 1002.267,A -85,B 0,C 180,E1 -13437.785,E2 -13437.785} C_VEL
LIN {X 0,Y 471.059,Z 987.73,A -85,B 0,C 180,E1 -13440.062,E2 -13440.062} C_VEL
LIN {X 0,Y 475.213,Z 971.011,A -85,B 0,C 180,E1 -13442.36,E2 -13442.36} C_VEL
LIN {X 0,Y 479.52,Z 953.243,A -85,B 0,C 180,E1 -13444.445,E2 -13444.445} C_VEL
LIN {X 0,Y 483.735,Z 935.751,A -85,B 0,C 180,E1 -13446.24,E2 -13446.24} C_VEL
LIN {X 0,Y 488.441,Z 915.324,A -85,B 0,C 180,E1 -13448.038,E2 -13448.038} C_VEL
LIN {X 0,Y 492.504,Z 896.616,A -85,B 0,C 180,E1 -13449.454,E2 -13449.454} C_VEL
LIN {X 0,Y 497.11,Z 873.76,A -85,B 0,C 180,E1 -13450.925,E2 -13450.925} C_VEL
LIN {X 0,Y 500.682,Z 853.949,A -85,B 0,C 180,E1 -13451.991,E2 -13451.991} C_VEL
LIN {X 0,Y 504.312,Z 831.603,A -85,B 0,C 180,E1 -13453.003,E2 -13453.003} C_VEL
LIN {X 0,Y 507.469,Z 808.093,A -85,B 0,C 180,E1 -13453.842,E2 -13453.842} C_VEL
LIN {X 0,Y 509.804,Z 787.373,A -85,B 0,C 180,E1 -13454.428,E2 -13454.428} C_VEL
LIN {X 0,Y 511.932,Z 760.897,A -85,B 0,C 180,E1 -13454.98,E2 -13454.98} C_VEL
LIN {X 0,Y 520.999,Z 535.801,A -85,B 0,C 180,E1 -13458.376,E2 -13458.376} C_VEL
LIN {X 0,Y 523.883,Z 463.407,A -85,B 0,C 180,E1 -13459.48,E2 -13459.48} C_VEL
LIN {X 0,Y 511.785,Z 442.286,A -85,B 0,C 180,E1 -13461.482,E2 -13461.482} C_VEL
LIN {X 0,Y 500.842,Z 424.786,A -85,B 0,C 180,E1 -13463.421,E2 -13463.421} C_VEL
LIN {X 0,Y 489.825,Z 408.153,A -85,B 0,C 180,E1 -13465.531,E2 -13465.531} C_VEL
LIN {X 0,Y 479.895,Z 394.334,A -85,B 0,C 180,E1 -13467.588,E2 -13467.588} C_VEL
LIN {X 0,Y 475.36,Z 388.159,A -85,B 0,C 180,E1 -13468.592,E2 -13468.592} C_VEL
LIN {X 0,Y 468.654,Z 379.399,A -85,B 0,C 180,E1 -13470.155,E2 -13470.155} C_VEL
LIN {X 0,Y 464.766,Z 374.244,A -85,B 0,C 180,E1 -13471.119,E2 -13471.119} C_VEL
LIN {X 0,Y 461.291,Z 369.861,A -85,B 0,C 180,E1 -13472.012,E2 -13472.012} C_VEL
LIN {X 0,Y 459.51,Z 367.643,A -85,B 0,C 180,E1 -13472.528,E2 -13472.528} C_VEL
LIN {X 0,Y 458.209,Z 364.129,A -85,B 0,C 180,E1 -13473.566,E2 -13473.566} C_VEL
LIN {X 0,Y 458.237,Z 364.121,A -85,B 0,C 180,E1 -13477.28,E2 -13477.28} C_VEL
LIN {X 0,Y 458.195,Z 364.124,A -85,B 0,C 180,E1 -13480.893,E2 -13480.893} C_VEL
LIN {X 0,Y 458.177,Z 364.139,A -85,B 0,C 180,E1 -13484.429,E2 -13484.429} C_VEL
LIN {X 0,Y 458.196,Z 364.158,A -85,B 0,C 180,E1 -13488.035,E2 -13488.035} C_VEL
LIN {X 0,Y 458.225,Z 364.127,A -85,B 0,C 180,E1 -13491.72,E2 -13491.72} C_VEL
LIN {X 0,Y 458.202,Z 364.12,A -85,B 0,C 180,E1 -13495.243,E2 -13495.243} C_VEL
LIN {X 0,Y 458.182,Z 364.151,A -85,B 0,C 180,E1 -13498.875,E2 -13498.875} C_VEL
LIN {X 0,Y 458.179,Z 364.147,A -85,B 0,C 180,E1 -13502.627,E2 -13502.627} C_VEL
LIN {X 0,Y 458.196,Z 364.119,A -85,B 0,C 180,E1 -13506.264,E2 -13506.264} C_VEL
LIN {X 0,Y 458.227,Z 364.131,A -85,B 0,C 180,E1 -13509.8,E2 -13509.8} C_VEL
LIN {X 0,Y 458.205,Z 364.154,A -85,B 0,C 180,E1 -13513.503,E2 -13513.503} C_VEL
LIN {X 0,Y 458.18,Z 364.131,A -85,B 0,C 180,E1 -13517.089,E2 -13517.089} C_VEL
LIN {X 0,Y 458.187,Z 364.124,A -85,B 0,C 180,E1 -13520.703,E2 -13520.703} C_VEL
LIN {X 0,Y 458.228,Z 364.132,A -85,B 0,C 180,E1 -13524.22,E2 -13524.22} C_VEL
LIN {X 0,Y 458.228,Z 364.144,A -85,B 0,C 180,E1 -13527.979,E2 -13527.979} C_VEL
LIN {X 0,Y 458.211,Z 364.286,A -85,B 0,C 180,E1 -13529.526,E2 -13529.526} C_VEL
LIN {X 0,Y 459.283,Z 367.238,A -85,B 0,C 180,E1 -13529.868,E2 -13529.868} C_VEL
LIN {X 0,Y 462.015,Z 369.995,A -85,B 0,C 180,E1 -13530.57,E2 -13530.57} C_VEL
LIN {X 0,Y 463.272,Z 370.893,A -85,B 0,C 180,E1 -13530.873,E2 -13530.873} C_VEL
LIN {X 0,Y 465.505,Z 374.546,A -85,B 0,C 180,E1 -13531.464,E2 -13531.464} C_VEL
LIN {X 0,Y 468.396,Z 377.252,A -85,B 0,C 180,E1 -13532.146,E2 -13532.146} C_VEL
LIN {X 0,Y 471.287,Z 381.231,A -85,B 0,C 180,E1 -13532.843,E2 -13532.843} C_VEL
LIN {X 0,Y 473.371,Z 383.378,A -85,B 0,C 180,E1 -13533.312,E2 -13533.312} C_VEL
LIN {X 0,Y 476.936,Z 387.841,A -85,B 0,C 180,E1 -13534.112,E2 -13534.112} C_VEL
LIN {X 0,Y 483.044,Z 395.643,A -85,B 0,C 180,E1 -13535.422,E2 -13535.422} C_VEL
LIN {X 0,Y 490.401,Z 405.035,A -85,B 0,C 180,E1 -13536.903,E2 -13536.903} C_VEL
LIN {X 0,Y 502.827,Z 421.982,A -85,B 0,C 180,E1 -13539.224,E2 -13539.224} C_VEL
LIN {X 0,Y 514.636,Z 439.254,A -85,B 0,C 180,E1 -13541.252,E2 -13541.252} C_VEL
LIN {X 0,Y 523.263,Z 453.508,A -85,B 0,C 180,E1 -13542.66,E2 -13542.66} C_VEL
LIN {X 0,Y 524.165,Z 455.483,A -85,B 0,C 180,E1 -13542.812,E2 -13542.812} C_VEL
LIN {X 0,Y 513.966,Z 706.066,A -85,B 0,C 180,E1 -13546.57,E2 -13546.57} C_VEL
LIN {X 0,Y 512.058,Z 747.8,A -85,B 0,C 180,E1 -13547.229,E2 -13547.229} C_VEL
LIN {X 0,Y 510.005,Z 771.636,A -85,B 0,C 180,E1 -13547.783,E2 -13547.783} C_VEL
LIN {X 0,Y 507.431,Z 795.134,A -85,B 0,C 180,E1 -13548.499,E2 -13548.499} C_VEL
LIN {X 0,Y 504.175,Z 818.329,A -85,B 0,C 180,E1 -13549.421,E2 -13549.421} C_VEL
LIN {X 0,Y 500.793,Z 839.443,A -85,B 0,C 180,E1 -13550.438,E2 -13550.438} C_VEL
LIN {X 0,Y 496.611,Z 861.877,A -85,B 0,C 180,E1 -13551.743,E2 -13551.743} C_VEL
LIN {X 0,Y 492.66,Z 881.26,A -85,B 0,C 180,E1 -13553.076,E2 -13553.076} C_VEL
LIN {X 0,Y 487.817,Z 902.979,A -85,B 0,C 180,E1 -13554.832,E2 -13554.832} C_VEL
LIN {X 0,Y 483.789,Z 919.932,A -85,B 0,C 180,E1 -13556.429,E2 -13556.429} C_VEL
LIN {X 0,Y 479.098,Z 938.966,A -85,B 0,C 180,E1 -13558.494,E2 -13558.494} C_VEL
LIN {X 0,Y 475.07,Z 954.781,A -85,B 0,C 180,E1 -13560.495,E2 -13560.495} C_VEL
LIN {X 0,Y 470.99,Z 971.03,A -85,B 0,C 180,E1 -13562.843,E2 -13562.843} C_VEL
LIN {X 0,Y 467.289,Z 985.698,A -85,B 0,C 180,E1 -13565.339,E2 -13565.339} C_VEL
LIN {X 0,Y 464.096,Z 999.223,A -85,B 0,C 180,E1 -13567.983,E2 -13567.983} C_VEL
LIN {X 0,Y 462.054,Z 1008.223,A -85,B 0,C 180,E1 -13570.027,E2 -13570.027} C_VEL
LIN {X 0,Y 460.335,Z 1011.752,A -85,B 0,C 180,E1 -13570.862,E2 -13570.862} C_VEL
LIN {X 0,Y 452.501,Z 1020.938,A -85,B 0,C 180,E1 -13573.06,E2 -13573.06} C_VEL
LIN {X 0,Y 451.27,Z 1023.48,A -85,B 0,C 180,E1 -13573.824,E2 -13573.824} C_VEL
LIN {X 0,Y 449.909,Z 1031.245,A -85,B 0,C 180,E1 -13576.505,E2 -13576.505} C_VEL
LIN {X 0,Y 448.891,Z 1038.635,A -85,B 0,C 180,E1 -13579.606,E2 -13579.606} C_VEL
LIN {X 0,Y 448.318,Z 1043.981,A -85,B 0,C 180,E1 -13582.568,E2 -13582.568} C_VEL
LIN {X 0,Y 448.067,Z 1047.8,A -85,B 0,C 180,E1 -13585.392,E2 -13585.392} C_VEL
LIN {X 0,Y 447.969,Z 1050.386,A -85,B 0,C 180,E1 -13588.465,E2 -13588.465} C_VEL
LIN {X 0,Y 447.946,Z 1051.365,A -85,B 0,C 180,E1 -13591.023,E2 -13591.023} C_VEL
LIN {X 0,Y 447.945,Z 1051.286,A -85,B 0,C 180,E1 -13593.712,E2 -13593.712} C_VEL
LIN {X 0,Y 448.003,Z 1049.625,A -85,B 0,C 180,E1 -13596.922,E2 -13596.922} C_VEL
LIN {X 0,Y 448.14,Z 1046.892,A -85,B 0,C 180,E1 -13599.633,E2 -13599.633} C_VEL
LIN {X 0,Y 448.485,Z 1042.782,A -85,B 0,C 180,E1 -13602.489,E2 -13602.489} C_VEL
LIN {X 0,Y 449.242,Z 1036.576,A -85,B 0,C 180,E1 -13605.623,E2 -13605.623} C_VEL
LIN {X 0,Y 450.334,Z 1029.744,A -85,B 0,C 180,E1 -13608.378,E2 -13608.378} C_VEL
LIN {X 0,Y 452.29,Z 1019.684,A -85,B 0,C 180,E1 -13611.666,E2 -13611.666} C_VEL
LIN {X 0,Y 454.442,Z 1010.029,A -85,B 0,C 180,E1 -13614.296,E2 -13614.296} C_VEL
LIN {X 0,Y 457.697,Z 996.962,A -85,B 0,C 180,E1 -13617.308,E2 -13617.308} C_VEL
LIN {X 0,Y 460.846,Z 985.072,A -85,B 0,C 180,E1 -13619.649,E2 -13619.649} C_VEL
LIN {X 0,Y 465.013,Z 970.007,A -85,B 0,C 180,E1 -13622.226,E2 -13622.226} C_VEL
LIN {X 0,Y 469.151,Z 954.945,A -85,B 0,C 180,E1 -13624.431,E2 -13624.431} C_VEL
LIN {X 0,Y 474.018,Z 937.548,A -85,B 0,C 180,E1 -13626.652,E2 -13626.652} C_VEL
LIN {X 0,Y 478.863,Z 919.276,A -85,B 0,C 180,E1 -13628.633,E2 -13628.633} C_VEL
LIN {X 0,Y 483.509,Z 901.231,A -85,B 0,C 180,E1 -13630.337,E2 -13630.337} C_VEL
LIN {X 0,Y 488.483,Z 880.317,A -85,B 0,C 180,E1 -13632.017,E2 -13632.017} C_VEL
LIN {X 0,Y 492.633,Z 861.423,A -85,B 0,C 180,E1 -13633.317,E2 -13633.317} C_VEL
LIN {X 0,Y 497.429,Z 837.175,A -85,B 0,C 180,E1 -13634.712,E2 -13634.712} C_VEL
LIN {X 0,Y 500.905,Z 816.856,A -85,B 0,C 180,E1 -13635.68,E2 -13635.68} C_VEL
LIN {X 0,Y 504.59,Z 791.469,A -85,B 0,C 180,E1 -13636.656,E2 -13636.656} C_VEL
LIN {X 0,Y 507.126,Z 769.58,A -85,B 0,C 180,E1 -13637.307,E2 -13637.307} C_VEL
LIN {X 0,Y 509.367,Z 743.567,A -85,B 0,C 180,E1 -13637.877,E2 -13637.877} C_VEL
LIN {X 0,Y 514.182,Z 636.144,A -85,B 0,C 180,E1 -13639.527,E2 -13639.527} C_VEL
LIN {X 0,Y 522.059,Z 460.243,A -85,B 0,C 180,E1 -13642.201,E2 -13642.201} C_VEL
LIN {X 0,Y 513.94,Z 447.186,A -85,B 0,C 180,E1 -13643.636,E2 -13643.636} C_VEL
LIN {X 0,Y 502.833,Z 431.077,A -85,B 0,C 180,E1 -13645.719,E2 -13645.719} C_VEL
LIN {X 0,Y 492.123,Z 416.54,A -85,B 0,C 180,E1 -13647.906,E2 -13647.906} C_VEL
LIN {X 0,Y 483.349,Z 405.363,A -85,B 0,C 180,E1 -13649.856,E2 -13649.856} C_VEL
LIN {X 0,Y 479.641,Z 400.723,A -85,B 0,C 180,E1 -13650.735,E2 -13650.735} C_VEL
LIN {X 0,Y 475.383,Z 395.471,A -85,B 0,C 180,E1 -13651.788,E2 -13651.788} C_VEL
LIN {X 0,Y 471.694,Z 390.827,A -85,B 0,C 180,E1 -13652.75,E2 -13652.75} C_VEL
LIN {X 0,Y 467.461,Z 386.141,A -85,B 0,C 180,E1 -13653.89,E2 -13653.89} C_VEL
LIN {X 0,Y 465.998,Z 384.075,A -85,B 0,C 180,E1 -13654.314,E2 -13654.314} C_VEL
LIN {X 0,Y 462.725,Z 380.846,A -85,B 0,C 180,E1 -13655.249,E2 -13655.249} C_VEL
LIN {X 0,Y 461,Z 378.066,A -85,B 0,C 180,E1 -13655.799,E2 -13655.799} C_VEL
LIN {X 0,Y 457.667,Z 375.328,A -85,B 0,C 180,E1 -13656.809,E2 -13656.809} C_VEL
LIN {X 0,Y 455.565,Z 371.69,A -85,B 0,C 180,E1 -13657.548,E2 -13657.548} C_VEL
LIN {X 0,Y 452.317,Z 369.569,A -85,B 0,C 180,E1 -13658.608,E2 -13658.608} C_VEL
LIN {X 0,Y 450.629,Z 366.764,A -85,B 0,C 180,E1 -13659.256,E2 -13659.256} C_VEL
LIN {X 0,Y 450.258,Z 365.131,A -85,B 0,C 180,E1 -13659.459,E2 -13659.459} C_VEL
LIN {X 0,Y 450.24,Z 365.13,A -85,B 0,C 180,E1 -13663.087,E2 -13663.087} C_VEL
LIN {X 0,Y 450.245,Z 365.125,A -85,B 0,C 180,E1 -13666.777,E2 -13666.777} C_VEL
LIN {X 0,Y 450.274,Z 365.117,A -85,B 0,C 180,E1 -13670.413,E2 -13670.413} C_VEL
LIN {X 0,Y 450.281,Z 365.115,A -85,B 0,C 180,E1 -13674.009,E2 -13674.009} C_VEL
LIN {X 0,Y 450.244,Z 365.128,A -85,B 0,C 180,E1 -13677.582,E2 -13677.582} C_VEL
LIN {X 0,Y 450.242,Z 365.141,A -85,B 0,C 180,E1 -13681.273,E2 -13681.273} C_VEL
LIN {X 0,Y 450.254,Z 365.147,A -85,B 0,C 180,E1 -13684.969,E2 -13684.969} C_VEL
LIN {X 0,Y 450.289,Z 365.128,A -85,B 0,C 180,E1 -13688.556,E2 -13688.556} C_VEL
LIN {X 0,Y 450.277,Z 365.12,A -85,B 0,C 180,E1 -13692.309,E2 -13692.309} C_VEL
LIN {X 0,Y 450.242,Z 365.118,A -85,B 0,C 180,E1 -13695.852,E2 -13695.852} C_VEL
LIN {X 0,Y 450.236,Z 365.118,A -85,B 0,C 180,E1 -13699.593,E2 -13699.593} C_VEL
LIN {X 0,Y 450.27,Z 365.319,A -85,B 0,C 180,E1 -13701.974,E2 -13701.974} C_VEL
LIN {X 0,Y 450.835,Z 367.205,A -85,B 0,C 180,E1 -13702.494,E2 -13702.494} C_VEL
LIN {X 0,Y 452.772,Z 370.012,A -85,B 0,C 180,E1 -13703.216,E2 -13703.216} C_VEL
LIN {X 0,Y 455.076,Z 371.943,A -85,B 0,C 180,E1 -13703.984,E2 -13703.984} C_VEL
LIN {X 0,Y 460.359,Z 378.534,A -85,B 0,C 180,E1 -13705.712,E2 -13705.712} C_VEL
LIN {X 0,Y 464.269,Z 383.156,A -85,B 0,C 180,E1 -13706.89,E2 -13706.89} C_VEL
LIN {X 0,Y 468.019,Z 387.859,A -85,B 0,C 180,E1 -13707.966,E2 -13707.966} C_VEL
LIN {X 0,Y 476.867,Z 399.572,A -85,B 0,C 180,E1 -13710.318,E2 -13710.318} C_VEL
LIN {X 0,Y 485.216,Z 410.905,A -85,B 0,C 180,E1 -13712.327,E2 -13712.327} C_VEL
LIN {X 0,Y 493.768,Z 423.223,A -85,B 0,C 180,E1 -13714.226,E2 -13714.226} C_VEL
LIN {X 0,Y 501.974,Z 435.595,A -85,B 0,C 180,E1 -13715.918,E2 -13715.918} C_VEL
LIN {X 0,Y 512.044,Z 451.745,A -85,B 0,C 180,E1 -13717.854,E2 -13717.854} C_VEL
LIN {X 0,Y 521.934,Z 468.785,A -85,B 0,C 180,E1 -13719.632,E2 -13719.632} C_VEL
LIN {X 0,Y 511.106,Z 713.472,A -85,B 0,C 180,E1 -13723.343,E2 -13723.343} C_VEL
LIN {X 0,Y 508.654,Z 765.631,A -85,B 0,C 180,E1 -13724.162,E2 -13724.162} C_VEL
LIN {X 0,Y 506.312,Z 790.128,A -85,B 0,C 180,E1 -13724.708,E2 -13724.708} C_VEL
LIN {X 0,Y 503.745,Z 810.967,A -85,B 0,C 180,E1 -13725.315,E2 -13725.315} C_VEL
LIN {X 0,Y 500.065,Z 835.287,A -85,B 0,C 180,E1 -13726.225,E2 -13726.225} C_VEL
LIN {X 0,Y 496.645,Z 854.769,A -85,B 0,C 180,E1 -13727.125,E2 -13727.125} C_VEL
LIN {X 0,Y 492.202,Z 877.43,A -85,B 0,C 180,E1 -13728.372,E2 -13728.372} C_VEL
LIN {X 0,Y 487.577,Z 898.273,A -85,B 0,C 180,E1 -13729.761,E2 -13729.761} C_VEL
LIN {X 0,Y 482.825,Z 918.479,A -85,B 0,C 180,E1 -13731.328,E2 -13731.328} C_VEL
LIN {X 0,Y 477.745,Z 938.393,A -85,B 0,C 180,E1 -13733.157,E2 -13733.157} C_VEL
LIN {X 0,Y 473.211,Z 955.74,A -85,B 0,C 180,E1 -13734.993,E2 -13734.993} C_VEL
LIN {X 0,Y 468.212,Z 974.396,A -85,B 0,C 180,E1 -13737.296,E2 -13737.296} C_VEL
LIN {X 0,Y 464.166,Z 989.477,A -85,B 0,C 180,E1 -13739.444,E2 -13739.444} C_VEL
LIN {X 0,Y 459.907,Z 1005.746,A -85,B 0,C 180,E1 -13742.132,E2 -13742.132} C_VEL
LIN {X 0,Y 456.712,Z 1018.542,A -85,B 0,C 180,E1 -13744.589,E2 -13744.589} C_VEL
LIN {X 0,Y 453.523,Z 1032.445,A -85,B 0,C 180,E1 -13747.715,E2 -13747.715} C_VEL
LIN {X 0,Y 451.526,Z 1042.299,A -85,B 0,C 180,E1 -13750.33,E2 -13750.33} C_VEL
LIN {X 0,Y 449.832,Z 1052.269,A -85,B 0,C 180,E1 -13753.47,E2 -13753.47} C_VEL
LIN {X 0,Y 448.876,Z 1059.387,A -85,B 0,C 180,E1 -13756.219,E2 -13756.219} C_VEL
LIN {X 0,Y 448.274,Z 1065.688,A -85,B 0,C 180,E1 -13759.201,E2 -13759.201} C_VEL
LIN {X 0,Y 447.995,Z 1070.282,A -85,B 0,C 180,E1 -13762.175,E2 -13762.175} C_VEL
LIN {X 0,Y 447.945,Z 1073.099,A -85,B 0,C 180,E1 -13764.749,E2 -13764.749} C_VEL
LIN {X 0,Y 447.938,Z 1075.03,A -85,B 0,C 180,E1 -13767.697,E2 -13767.697} C_VEL
LIN {X 0,Y 447.939,Z 1075.344,A -85,B 0,C 180,E1 -13770.639,E2 -13770.639} C_VEL
LIN {X 0,Y 447.943,Z 1074.469,A -85,B 0,C 180,E1 -13773.199,E2 -13773.199} C_VEL
LIN {X 0,Y 447.955,Z 1072.272,A -85,B 0,C 180,E1 -13776.022,E2 -13776.022} C_VEL
LIN {X 0,Y 448.079,Z 1068.203,A -85,B 0,C 180,E1 -13779.116,E2 -13779.116} C_VEL
LIN {X 0,Y 448.424,Z 1063.366,A -85,B 0,C 180,E1 -13781.796,E2 -13781.796} C_VEL
LIN {X 0,Y 449.173,Z 1056.41,A -85,B 0,C 180,E1 -13784.833,E2 -13784.833} C_VEL
LIN {X 0,Y 450.365,Z 1048.003,A -85,B 0,C 180,E1 -13787.738,E2 -13787.738} C_VEL
LIN {X 0,Y 452.098,Z 1038.249,A -85,B 0,C 180,E1 -13790.589,E2 -13790.589} C_VEL
LIN {X 0,Y 454.492,Z 1026.41,A -85,B 0,C 180,E1 -13793.466,E2 -13793.466} C_VEL
LIN {X 0,Y 457.338,Z 1014.003,A -85,B 0,C 180,E1 -13796.069,E2 -13796.069} C_VEL
LIN {X 0,Y 461.01,Z 998.825,A -85,B 0,C 180,E1 -13798.783,E2 -13798.783} C_VEL
LIN {X 0,Y 464.563,Z 984.836,A -85,B 0,C 180,E1 -13800.958,E2 -13800.958} C_VEL
LIN {X 0,Y 469.251,Z 966.475,A -85,B 0,C 180,E1 -13803.423,E2 -13803.423} C_VEL
LIN {X 0,Y 473.301,Z 950.565,A -85,B 0,C 180,E1 -13805.269,E2 -13805.269} C_VEL
LIN {X 0,Y 478.374,Z 930.215,A -85,B 0,C 180,E1 -13807.312,E2 -13807.312} C_VEL
LIN {X 0,Y 482.676,Z 911.955,A -85,B 0,C 180,E1 -13808.879,E2 -13808.879} C_VEL
LIN {X 0,Y 487.326,Z 891.147,A -85,B 0,C 180,E1 -13810.428,E2 -13810.428} C_VEL
LIN {X 0,Y 491.661,Z 869.604,A -85,B 0,C 180,E1 -13811.762,E2 -13811.762} C_VEL
LIN {X 0,Y 495.61,Z 848.055,A -85,B 0,C 180,E1 -13812.893,E2 -13812.893} C_VEL
LIN {X 0,Y 499.32,Z 824.384,A -85,B 0,C 180,E1 -13813.897,E2 -13813.897} C_VEL
LIN {X 0,Y 502.316,Z 802.163,A -85,B 0,C 180,E1 -13814.651,E2 -13814.651} C_VEL
LIN {X 0,Y 504.985,Z 776.643,A -85,B 0,C 180,E1 -13815.303,E2 -13815.303} C_VEL
LIN {X 0,Y 506.564,Z 754.118,A -85,B 0,C 180,E1 -13815.724,E2 -13815.724} C_VEL
LIN {X 0,Y 516.933,Z 505.006,A -85,B 0,C 180,E1 -13819.495,E2 -13819.495} C_VEL
LIN {X 0,Y 518.425,Z 466.807,A -85,B 0,C 180,E1 -13820.093,E2 -13820.093} C_VEL
LIN {X 0,Y 506.72,Z 446.358,A -85,B 0,C 180,E1 -13822.09,E2 -13822.09} C_VEL
LIN {X 0,Y 496.467,Z 429.865,A -85,B 0,C 180,E1 -13823.96,E2 -13823.96} C_VEL
LIN {X 0,Y 486.048,Z 414.014,A -85,B 0,C 180,E1 -13826.01,E2 -13826.01} C_VEL
LIN {X 0,Y 476.62,Z 400.744,A -85,B 0,C 180,E1 -13828.014,E2 -13828.014} C_VEL
LIN {X 0,Y 470.189,Z 391.86,A -85,B 0,C 180,E1 -13829.488,E2 -13829.488} C_VEL
LIN {X 0,Y 465.532,Z 385.893,A -85,B 0,C 180,E1 -13830.608,E2 -13830.608} C_VEL
LIN {X 0,Y 461.918,Z 381.059,A -85,B 0,C 180,E1 -13831.526,E2 -13831.526} C_VEL
LIN {X 0,Y 456.914,Z 374.765,A -85,B 0,C 180,E1 -13832.853,E2 -13832.853} C_VEL
LIN {X 0,Y 453.412,Z 370.552,A -85,B 0,C 180,E1 -13833.829,E2 -13833.829} C_VEL
LIN {X 0,Y 451.1,Z 367.867,A -85,B 0,C 180,E1 -13834.496,E2 -13834.496} C_VEL
LIN {X 0,Y 450.288,Z 365.126,A -85,B 0,C 180,E1 -13835.259,E2 -13835.259} C_VEL
LIN {X 0,Y 450.26,Z 365.145,A -85,B 0,C 180,E1 -13838.858,E2 -13838.858} C_VEL
LIN {X 0,Y 450.242,Z 365.132,A -85,B 0,C 180,E1 -13842.554,E2 -13842.554} C_VEL
LIN {X 0,Y 450.24,Z 365.115,A -85,B 0,C 180,E1 -13846.254,E2 -13846.254} C_VEL
LIN {X 0,Y 450.274,Z 365.11,A -85,B 0,C 180,E1 -13849.767,E2 -13849.767} C_VEL
LIN {X 0,Y 450.299,Z 365.136,A -85,B 0,C 180,E1 -13853.498,E2 -13853.498} C_VEL
LIN {X 0,Y 450.259,Z 365.128,A -85,B 0,C 180,E1 -13857.2,E2 -13857.2} C_VEL
LIN {X 0,Y 450.236,Z 365.107,A -85,B 0,C 180,E1 -13860.763,E2 -13860.763} C_VEL
LIN {X 0,Y 450.246,Z 365.129,A -85,B 0,C 180,E1 -13864.458,E2 -13864.458} C_VEL
LIN {X 0,Y 450.282,Z 365.135,A -85,B 0,C 180,E1 -13868.042,E2 -13868.042} C_VEL
LIN {X 0,Y 450.284,Z 365.106,A -85,B 0,C 180,E1 -13871.788,E2 -13871.788} C_VEL
LIN {X 0,Y 450.249,Z 365.117,A -85,B 0,C 180,E1 -13875.324,E2 -13875.324} C_VEL
LIN {X 0,Y 450.245,Z 365.146,A -85,B 0,C 180,E1 -13878.919,E2 -13878.919} C_VEL
LIN {X 0,Y 450.26,Z 365.134,A -85,B 0,C 180,E1 -13882.593,E2 -13882.593} C_VEL
LIN {X 0,Y 450.29,Z 365.115,A -85,B 0,C 180,E1 -13886.225,E2 -13886.225} C_VEL
LIN {X 0,Y 450.287,Z 365.336,A -85,B 0,C 180,E1 -13887.625,E2 -13887.625} C_VEL
LIN {X 0,Y 451.296,Z 368.138,A -85,B 0,C 180,E1 -13887.98,E2 -13887.98} C_VEL
LIN {X 0,Y 453.847,Z 370.847,A -85,B 0,C 180,E1 -13888.704,E2 -13888.704} C_VEL
LIN {X 0,Y 455.527,Z 371.957,A -85,B 0,C 180,E1 -13889.145,E2 -13889.145} C_VEL
LIN {X 0,Y 457.684,Z 375.518,A -85,B 0,C 180,E1 -13889.767,E2 -13889.767} C_VEL
LIN {X 0,Y 460.657,Z 378.21,A -85,B 0,C 180,E1 -13890.525,E2 -13890.525} C_VEL
LIN {X 0,Y 463.451,Z 382.175,A -85,B 0,C 180,E1 -13891.257,E2 -13891.257} C_VEL
LIN {X 0,Y 465.734,Z 384.434,A -85,B 0,C 180,E1 -13891.808,E2 -13891.808} C_VEL
LIN {X 0,Y 469.137,Z 388.783,A -85,B 0,C 180,E1 -13892.631,E2 -13892.631} C_VEL
LIN {X 0,Y 470.884,Z 390.867,A -85,B 0,C 180,E1 -13893.038,E2 -13893.038} C_VEL
LIN {X 0,Y 476.097,Z 397.437,A -85,B 0,C 180,E1 -13894.217,E2 -13894.217} C_VEL
LIN {X 0,Y 480.36,Z 402.894,A -85,B 0,C 180,E1 -13895.138,E2 -13895.138} C_VEL
LIN {X 0,Y 487.396,Z 412.001,A -85,B 0,C 180,E1 -13896.581,E2 -13896.581} C_VEL
LIN {X 0,Y 499.444,Z 428.57,A -85,B 0,C 180,E1 -13898.876,E2 -13898.876} C_VEL
LIN {X 0,Y 511.635,Z 446.615,A -85,B 0,C 180,E1 -13901.008,E2 -13901.008} C_VEL
LIN {X 0,Y 518.739,Z 458.868,A -85,B 0,C 180,E1 -13902.2,E2 -13902.2} C_VEL
LIN {X 0,Y 508.149,Z 709.985,A -85,B 0,C 180,E1 -13905.992,E2 -13905.992} C_VEL
LIN {X 0,Y 506.28,Z 748.548,A -85,B 0,C 180,E1 -13906.612,E2 -13906.612} C_VEL
LIN {X 0,Y 504.192,Z 772.045,A -85,B 0,C 180,E1 -13907.162,E2 -13907.162} C_VEL
LIN {X 0,Y 501.494,Z 795.854,A -85,B 0,C 180,E1 -13907.895,E2 -13907.895} C_VEL
LIN {X 0,Y 498.135,Z 818.964,A -85,B 0,C 180,E1 -13908.823,E2 -13908.823} C_VEL
LIN {X 0,Y 494.465,Z 841.146,A -85,B 0,C 180,E1 -13909.905,E2 -13909.905} C_VEL
LIN {X 0,Y 490.296,Z 862.557,A -85,B 0,C 180,E1 -13911.173,E2 -13911.173} C_VEL
LIN {X 0,Y 486.249,Z 881.746,A -85,B 0,C 180,E1 -13912.506,E2 -13912.506} C_VEL
LIN {X 0,Y 481.239,Z 903.419,A -85,B 0,C 180,E1 -13914.279,E2 -13914.279} C_VEL
LIN {X 0,Y 477.113,Z 920.181,A -85,B 0,C 180,E1 -13915.874,E2 -13915.874} C_VEL
LIN {X 0,Y 472.225,Z 939.257,A -85,B 0,C 180,E1 -13917.967,E2 -13917.967} C_VEL
LIN {X 0,Y 468.005,Z 955.157,A -85,B 0,C 180,E1 -13920.004,E2 -13920.004} C_VEL
LIN {X 0,Y 463.735,Z 971.472,A -85,B 0,C 180,E1 -13922.398,E2 -13922.398} C_VEL
LIN {X 0,Y 459.89,Z 986.038,A -85,B 0,C 180,E1 -13924.915,E2 -13924.915} C_VEL
LIN {X 0,Y 456.552,Z 999.545,A -85,B 0,C 180,E1 -13927.6,E2 -13927.6} C_VEL
LIN {X 0,Y 453.842,Z 1010.974,A -85,B 0,C 180,E1 -13930.301,E2 -13930.301} C_VEL
LIN {X 0,Y 451.777,Z 1020.868,A -85,B 0,C 180,E1 -13933.013,E2 -13933.013} C_VEL
LIN {X 0,Y 451.27,Z 1023.48,A -85,B 0,C 180,E1 -13933.824,E2 -13933.824} C_VEL
LIN {X 0,Y 449.761,Z 1026.387,A -85,B 0,C 180,E1 -13934.722,E2 -13934.722} C_VEL
LIN {X 0,Y 442.431,Z 1033.675,A -85,B 0,C 180,E1 -13937.111,E2 -13937.111} C_VEL
LIN {X 0,Y 441.394,Z 1035.6,A -85,B 0,C 180,E1 -13937.926,E2 -13937.926} C_VEL
LIN {X 0,Y 440.648,Z 1041.384,A -85,B 0,C 180,E1 -13940.729,E2 -13940.729} C_VEL
LIN {X 0,Y 440.168,Z 1046.479,A -85,B 0,C 180,E1 -13944.002,E2 -13944.002} C_VEL
LIN {X 0,Y 440.009,Z 1049.381,A -85,B 0,C 180,E1 -13946.743,E2 -13946.743} C_VEL
LIN {X 0,Y 439.954,Z 1051.147,A -85,B 0,C 180,E1 -13949.479,E2 -13949.479} C_VEL
LIN {X 0,Y 439.94,Z 1051.693,A -85,B 0,C 180,E1 -13952.605,E2 -13952.605} C_VEL
LIN {X 0,Y 439.969,Z 1050.878,A -85,B 0,C 180,E1 -13955.346,E2 -13955.346} C_VEL
LIN {X 0,Y 440.043,Z 1049.04,A -85,B 0,C 180,E1 -13957.967,E2 -13957.967} C_VEL
LIN {X 0,Y 440.31,Z 1045.196,A -85,B 0,C 180,E1 -13961.262,E2 -13961.262} C_VEL
LIN {X 0,Y 440.816,Z 1040.543,A -85,B 0,C 180,E1 -13964.046,E2 -13964.046} C_VEL
LIN {X 0,Y 441.744,Z 1034.349,A -85,B 0,C 180,E1 -13966.977,E2 -13966.977} C_VEL
LIN {X 0,Y 443.258,Z 1026.119,A -85,B 0,C 180,E1 -13970.052,E2 -13970.052} C_VEL
LIN {X 0,Y 445.115,Z 1017.55,A -85,B 0,C 180,E1 -13972.729,E2 -13972.729} C_VEL
LIN {X 0,Y 448.164,Z 1005.199,A -85,B 0,C 180,E1 -13975.956,E2 -13975.956} C_VEL
LIN {X 0,Y 451.208,Z 993.916,A -85,B 0,C 180,E1 -13978.454,E2 -13978.454} C_VEL
LIN {X 0,Y 455.553,Z 978.507,A -85,B 0,C 180,E1 -13981.371,E2 -13981.371} C_VEL
LIN {X 0,Y 459.705,Z 964.184,A -85,B 0,C 180,E1 -13983.686,E2 -13983.686} C_VEL
LIN {X 0,Y 465.039,Z 945.702,A -85,B 0,C 180,E1 -13986.248,E2 -13986.248} C_VEL
LIN {X 0,Y 469.537,Z 929.823,A -85,B 0,C 180,E1 -13988.138,E2 -13988.138} C_VEL
LIN {X 0,Y 475.157,Z 909.241,A -85,B 0,C 180,E1 -13990.243,E2 -13990.243} C_VEL
LIN {X 0,Y 479.806,Z 891.095,A -85,B 0,C 180,E1 -13991.825,E2 -13991.825} C_VEL
LIN {X 0,Y 484.96,Z 869.463,A -85,B 0,C 180,E1 -13993.441,E2 -13993.441} C_VEL
LIN {X 0,Y 489.182,Z 849.717,A -85,B 0,C 180,E1 -13994.679,E2 -13994.679} C_VEL
LIN {X 0,Y 493.411,Z 827.942,A -85,B 0,C 180,E1 -13995.838,E2 -13995.838} C_VEL
LIN {X 0,Y 497.108,Z 805.082,A -85,B 0,C 180,E1 -13996.822,E2 -13996.822} C_VEL
LIN {X 0,Y 499.914,Z 784.791,A -85,B 0,C 180,E1 -13997.533,E2 -13997.533} C_VEL
LIN {X 0,Y 502.662,Z 759.493,A -85,B 0,C 180,E1 -13998.216,E2 -13998.216} C_VEL
LIN {X 0,Y 504.28,Z 737.69,A -85,B 0,C 180,E1 -13998.644,E2 -13998.644} C_VEL
LIN {X 0,Y 515.705,Z 490.195,A -85,B 0,C 180,E1 -14002.428,E2 -14002.428} C_VEL
LIN {X 0,Y 516.812,Z 463.843,A -85,B 0,C 180,E1 -14002.852,E2 -14002.852} C_VEL
LIN {X 0,Y 508.755,Z 450.942,A -85,B 0,C 180,E1 -14004.322,E2 -14004.322} C_VEL
LIN {X 0,Y 496.361,Z 433.111,A -85,B 0,C 180,E1 -14006.74,E2 -14006.74} C_VEL
LIN {X 0,Y 485.835,Z 418.911,A -85,B 0,C 180,E1 -14009,E2 -14009} C_VEL
LIN {X 0,Y 476.902,Z 407.617,A -85,B 0,C 180,E1 -14011.1,E2 -14011.1} C_VEL
LIN {X 0,Y 472.696,Z 402.404,A -85,B 0,C 180,E1 -14012.163,E2 -14012.163} C_VEL
LIN {X 0,Y 468.223,Z 396.919,A -85,B 0,C 180,E1 -14013.355,E2 -14013.355} C_VEL
LIN {X 0,Y 464.612,Z 392.56,A -85,B 0,C 180,E1 -14014.369,E2 -14014.369} C_VEL
LIN {X 0,Y 463.434,Z 391.165,A -85,B 0,C 180,E1 -14014.71,E2 -14014.71} C_VEL
LIN {X 0,Y 460.056,Z 387.445,A -85,B 0,C 180,E1 -14015.712,E2 -14015.712} C_VEL
LIN {X 0,Y 458.701,Z 385.415,A -85,B 0,C 180,E1 -14016.149,E2 -14016.149} C_VEL
LIN {X 0,Y 455.354,Z 382.348,A -85,B 0,C 180,E1 -14017.197,E2 -14017.197} C_VEL
LIN {X 0,Y 453.524,Z 379.251,A -85,B 0,C 180,E1 -14017.852,E2 -14017.852} C_VEL
LIN {X 0,Y 450.179,Z 376.741,A -85,B 0,C 180,E1 -14018.979,E2 -14018.979} C_VEL
LIN {X 0,Y 448.267,Z 373.433,A -85,B 0,C 180,E1 -14019.739,E2 -14019.739} C_VEL
LIN {X 0,Y 447.894,Z 372.768,A -85,B 0,C 180,E1 -14019.892,E2 -14019.892} C_VEL
LIN {X 0,Y 444.635,Z 370.837,A -85,B 0,C 180,E1 -14021.105,E2 -14021.105} C_VEL
LIN {X 0,Y 442.875,Z 368.133,A -85,B 0,C 180,E1 -14021.88,E2 -14021.88} C_VEL
LIN {X 0,Y 442.338,Z 366.106,A -85,B 0,C 180,E1 -14022.232,E2 -14022.232} C_VEL
LIN {X 0,Y 442.359,Z 366.102,A -85,B 0,C 180,E1 -14026.004,E2 -14026.004} C_VEL
LIN {X 0,Y 442.321,Z 366.108,A -85,B 0,C 180,E1 -14029.713,E2 -14029.713} C_VEL
LIN {X 0,Y 442.3,Z 366.118,A -85,B 0,C 180,E1 -14033.249,E2 -14033.249} C_VEL
LIN {X 0,Y 442.306,Z 366.128,A -85,B 0,C 180,E1 -14037.02,E2 -14037.02} C_VEL
LIN {X 0,Y 442.335,Z 366.134,A -85,B 0,C 180,E1 -14040.648,E2 -14040.648} C_VEL
LIN {X 0,Y 442.347,Z 366.12,A -85,B 0,C 180,E1 -14044.408,E2 -14044.408} C_VEL
LIN {X 0,Y 442.325,Z 366.11,A -85,B 0,C 180,E1 -14048.063,E2 -14048.063} C_VEL
LIN {X 0,Y 442.302,Z 366.107,A -85,B 0,C 180,E1 -14051.739,E2 -14051.739} C_VEL
LIN {X 0,Y 442.299,Z 366.106,A -85,B 0,C 180,E1 -14055.472,E2 -14055.472} C_VEL
LIN {X 0,Y 442.314,Z 366.105,A -85,B 0,C 180,E1 -14059.134,E2 -14059.134} C_VEL
LIN {X 0,Y 442.322,Z 366.277,A -85,B 0,C 180,E1 -14059.484,E2 -14059.484} C_VEL
LIN {X 0,Y 443.214,Z 368.939,A -85,B 0,C 180,E1 -14059.951,E2 -14059.951} C_VEL
LIN {X 0,Y 445.677,Z 371.68,A -85,B 0,C 180,E1 -14060.968,E2 -14060.968} C_VEL
LIN {X 0,Y 448.061,Z 373.157,A -85,B 0,C 180,E1 -14061.846,E2 -14061.846} C_VEL
LIN {X 0,Y 450.632,Z 377.217,A -85,B 0,C 180,E1 -14062.849,E2 -14062.849} C_VEL
LIN {X 0,Y 453.238,Z 379.579,A -85,B 0,C 180,E1 -14063.742,E2 -14063.742} C_VEL
LIN {X 0,Y 458.645,Z 386.423,A -85,B 0,C 180,E1 -14065.538,E2 -14065.538} C_VEL
LIN {X 0,Y 461.948,Z 390.347,A -85,B 0,C 180,E1 -14066.55,E2 -14066.55} C_VEL
LIN {X 0,Y 467.029,Z 396.989,A -85,B 0,C 180,E1 -14068.031,E2 -14068.031} C_VEL
LIN {X 0,Y 474.172,Z 406.465,A -85,B 0,C 180,E1 -14069.95,E2 -14069.95} C_VEL
LIN {X 0,Y 482.866,Z 418.454,A -85,B 0,C 180,E1 -14072.083,E2 -14072.083} C_VEL
LIN {X 0,Y 490.981,Z 430.365,A -85,B 0,C 180,E1 -14073.918,E2 -14073.918} C_VEL
LIN {X 0,Y 498.672,Z 442.104,A -85,B 0,C 180,E1 -14075.537,E2 -14075.537} C_VEL
LIN {X 0,Y 508.434,Z 457.967,A -85,B 0,C 180,E1 -14077.458,E2 -14077.458} C_VEL
LIN {X 0,Y 516.756,Z 472.571,A -85,B 0,C 180,E1 -14078.998,E2 -14078.998} C_VEL
LIN {X 0,Y 505.459,Z 719.112,A -85,B 0,C 180,E1 -14082.761,E2 -14082.761} C_VEL
LIN {X 0,Y 503.141,Z 765.997,A -85,B 0,C 180,E1 -14083.506,E2 -14083.506} C_VEL
LIN {X 0,Y 500.731,Z 790.293,A -85,B 0,C 180,E1 -14084.054,E2 -14084.054} C_VEL
LIN {X 0,Y 498.012,Z 811.651,A -85,B 0,C 180,E1 -14084.682,E2 -14084.682} C_VEL
LIN {X 0,Y 494.284,Z 835.385,A -85,B 0,C 180,E1 -14085.579,E2 -14085.579} C_VEL
LIN {X 0,Y 490.661,Z 855.328,A -85,B 0,C 180,E1 -14086.508,E2 -14086.508} C_VEL
LIN {X 0,Y 485.976,Z 878.276,A -85,B 0,C 180,E1 -14087.791,E2 -14087.791} C_VEL
LIN {X 0,Y 481.392,Z 898.253,A -85,B 0,C 180,E1 -14089.135,E2 -14089.135} C_VEL
LIN {X 0,Y 476.571,Z 918.04,A -85,B 0,C 180,E1 -14090.682,E2 -14090.682} C_VEL
LIN {X 0,Y 471.365,Z 937.738,A -85,B 0,C 180,E1 -14092.5,E2 -14092.5} C_VEL
LIN {X 0,Y 466.637,Z 955.097,A -85,B 0,C 180,E1 -14094.35,E2 -14094.35} C_VEL
LIN {X 0,Y 461.543,Z 973.356,A -85,B 0,C 180,E1 -14096.615,E2 -14096.615} C_VEL
LIN {X 0,Y 457.296,Z 988.506,A -85,B 0,C 180,E1 -14098.788,E2 -14098.788} C_VEL
LIN {X 0,Y 452.79,Z 1004.901,A -85,B 0,C 180,E1 -14101.511,E2 -14101.511} C_VEL
LIN {X 0,Y 449.393,Z 1017.799,A -85,B 0,C 180,E1 -14104.013,E2 -14104.013} C_VEL
LIN {X 0,Y 446.251,Z 1030.721,A -85,B 0,C 180,E1 -14106.914,E2 -14106.914} C_VEL
LIN {X 0,Y 443.949,Z 1041.201,A -85,B 0,C 180,E1 -14109.705,E2 -14109.705} C_VEL
LIN {X 0,Y 442.159,Z 1051.012,A -85,B 0,C 180,E1 -14112.768,E2 -14112.768} C_VEL
LIN {X 0,Y 440.987,Z 1058.875,A -85,B 0,C 180,E1 -14115.825,E2 -14115.825} C_VEL
LIN {X 0,Y 440.343,Z 1064.981,A -85,B 0,C 180,E1 -14118.739,E2 -14118.739} C_VEL
LIN {X 0,Y 440.015,Z 1069.92,A -85,B 0,C 180,E1 -14121.901,E2 -14121.901} C_VEL
LIN {X 0,Y 439.947,Z 1072.8,A -85,B 0,C 180,E1 -14124.545,E2 -14124.545} C_VEL
LIN {X 0,Y 439.94,Z 1074.616,A -85,B 0,C 180,E1 -14127.264,E2 -14127.264} C_VEL
LIN {X 0,Y 439.941,Z 1075.173,A -85,B 0,C 180,E1 -14130.391,E2 -14130.391} C_VEL
LIN {X 0,Y 439.945,Z 1074.317,A -85,B 0,C 180,E1 -14133.127,E2 -14133.127} C_VEL
LIN {X 0,Y 439.954,Z 1072.278,A -85,B 0,C 180,E1 -14135.87,E2 -14135.87} C_VEL
LIN {X 0,Y 440.072,Z 1068.387,A -85,B 0,C 180,E1 -14139.02,E2 -14139.02} C_VEL
LIN {X 0,Y 440.422,Z 1063.558,A -85,B 0,C 180,E1 -14141.79,E2 -14141.79} C_VEL
LIN {X 0,Y 441.131,Z 1057.143,A -85,B 0,C 180,E1 -14144.706,E2 -14144.706} C_VEL
LIN {X 0,Y 442.378,Z 1048.656,A -85,B 0,C 180,E1 -14147.766,E2 -14147.766} C_VEL
LIN {X 0,Y 444.002,Z 1039.698,A -85,B 0,C 180,E1 -14150.473,E2 -14150.473} C_VEL
LIN {X 0,Y 446.636,Z 1027.29,A -85,B 0,C 180,E1 -14153.624,E2 -14153.624} C_VEL
LIN {X 0,Y 449.397,Z 1015.646,A -85,B 0,C 180,E1 -14156.138,E2 -14156.138} C_VEL
LIN {X 0,Y 453.148,Z 1000.861,A -85,B 0,C 180,E1 -14158.897,E2 -14158.897} C_VEL
LIN {X 0,Y 456.994,Z 986.23,A -85,B 0,C 180,E1 -14161.235,E2 -14161.235} C_VEL
LIN {X 0,Y 461.561,Z 969.219,A -85,B 0,C 180,E1 -14163.607,E2 -14163.607} C_VEL
LIN {X 0,Y 466.175,Z 951.698,A -85,B 0,C 180,E1 -14165.691,E2 -14165.691} C_VEL
LIN {X 0,Y 471.19,Z 932.534,A -85,B 0,C 180,E1 -14167.673,E2 -14167.673} C_VEL
LIN {X 0,Y 475.946,Z 913.043,A -85,B 0,C 180,E1 -14169.38,E2 -14169.38} C_VEL
LIN {X 0,Y 480.325,Z 894.144,A -85,B 0,C 180,E1 -14170.818,E2 -14170.818} C_VEL
LIN {X 0,Y 485.174,Z 871.29,A -85,B 0,C 180,E1 -14172.28,E2 -14172.28} C_VEL
LIN {X 0,Y 489.097,Z 850.681,A -85,B 0,C 180,E1 -14173.386,E2 -14173.386} C_VEL
LIN {X 0,Y 493.287,Z 825.279,A -85,B 0,C 180,E1 -14174.495,E2 -14174.495} C_VEL
LIN {X 0,Y 496.275,Z 803.926,A -85,B 0,C 180,E1 -14175.232,E2 -14175.232} C_VEL
LIN {X 0,Y 499.179,Z 777.589,A -85,B 0,C 180,E1 -14175.924,E2 -14175.924} C_VEL
LIN {X 0,Y 500.827,Z 755.22,A -85,B 0,C 180,E1 -14176.35,E2 -14176.35} C_VEL
LIN {X 0,Y 511.526,Z 507.68,A -85,B 0,C 180,E1 -14180.126,E2 -14180.126} C_VEL
LIN {X 0,Y 513.043,Z 470.309,A -85,B 0,C 180,E1 -14180.716,E2 -14180.716} C_VEL
LIN {X 0,Y 502.048,Z 450.985,A -85,B 0,C 180,E1 -14182.649,E2 -14182.649} C_VEL
LIN {X 0,Y 490.607,Z 432.404,A -85,B 0,C 180,E1 -14184.812,E2 -14184.812} C_VEL
LIN {X 0,Y 478.766,Z 414.63,A -85,B 0,C 180,E1 -14187.254,E2 -14187.254} C_VEL
LIN {X 0,Y 467.489,Z 398.866,A -85,B 0,C 180,E1 -14189.826,E2 -14189.826} C_VEL
LIN {X 0,Y 458.988,Z 387.726,A -85,B 0,C 180,E1 -14191.965,E2 -14191.965} C_VEL
LIN {X 0,Y 454.272,Z 381.695,A -85,B 0,C 180,E1 -14193.248,E2 -14193.248} C_VEL
LIN {X 0,Y 451.019,Z 377.76,A -85,B 0,C 180,E1 -14194.174,E2 -14194.174} C_VEL
LIN {X 0,Y 448.461,Z 374.594,A -85,B 0,C 180,E1 -14194.936,E2 -14194.936} C_VEL
LIN {X 0,Y 446.748,Z 372.301,A -85,B 0,C 180,E1 -14195.469,E2 -14195.469} C_VEL
LIN {X 0,Y 443.911,Z 370.013,A -85,B 0,C 180,E1 -14196.328,E2 -14196.328} C_VEL
LIN {X 0,Y 442.519,Z 367.142,A -85,B 0,C 180,E1 -14196.831,E2 -14196.831} C_VEL
LIN {X 0,Y 442.344,Z 366.098,A -85,B 0,C 180,E1 -14197.12,E2 -14197.12} C_VEL
LIN {X 0,Y 442.308,Z 366.102,A -85,B 0,C 180,E1 -14200.728,E2 -14200.728} C_VEL
LIN {X 0,Y 442.3,Z 366.115,A -85,B 0,C 180,E1 -14204.394,E2 -14204.394} C_VEL
LIN {X 0,Y 442.32,Z 366.136,A -85,B 0,C 180,E1 -14207.996,E2 -14207.996} C_VEL
LIN {X 0,Y 442.348,Z 366.102,A -85,B 0,C 180,E1 -14211.682,E2 -14211.682} C_VEL
LIN {X 0,Y 442.33,Z 366.094,A -85,B 0,C 180,E1 -14215.332,E2 -14215.332} C_VEL
LIN {X 0,Y 442.307,Z 366.123,A -85,B 0,C 180,E1 -14218.964,E2 -14218.964} C_VEL
LIN {X 0,Y 442.302,Z 366.125,A -85,B 0,C 180,E1 -14222.721,E2 -14222.721} C_VEL
LIN {X 0,Y 442.305,Z 366.098,A -85,B 0,C 180,E1 -14226.49,E2 -14226.49} C_VEL
LIN {X 0,Y 442.341,Z 366.102,A -85,B 0,C 180,E1 -14230.024,E2 -14230.024} C_VEL
LIN {X 0,Y 442.36,Z 366.13,A -85,B 0,C 180,E1 -14233.863,E2 -14233.863} C_VEL
LIN {X 0,Y 442.33,Z 366.113,A -85,B 0,C 180,E1 -14237.632,E2 -14237.632} C_VEL
LIN {X 0,Y 442.304,Z 366.101,A -85,B 0,C 180,E1 -14241.205,E2 -14241.205} C_VEL
LIN {X 0,Y 442.305,Z 366.104,A -85,B 0,C 180,E1 -14244.972,E2 -14244.972} C_VEL
LIN {X 0,Y 442.339,Z 366.294,A -85,B 0,C 180,E1 -14245.501,E2 -14245.501} C_VEL
LIN {X 0,Y 443.294,Z 369.02,A -85,B 0,C 180,E1 -14245.878,E2 -14245.878} C_VEL
LIN {X 0,Y 445.743,Z 371.73,A -85,B 0,C 180,E1 -14246.657,E2 -14246.657} C_VEL
LIN {X 0,Y 447.768,Z 373.027,A -85,B 0,C 180,E1 -14247.244,E2 -14247.244} C_VEL
LIN {X 0,Y 449.926,Z 376.626,A -85,B 0,C 180,E1 -14247.928,E2 -14247.928} C_VEL
LIN {X 0,Y 453.113,Z 379.439,A -85,B 0,C 180,E1 -14248.815,E2 -14248.815} C_VEL
LIN {X 0,Y 455.896,Z 383.357,A -85,B 0,C 180,E1 -14249.606,E2 -14249.606} C_VEL
LIN {X 0,Y 458.238,Z 385.663,A -85,B 0,C 180,E1 -14250.218,E2 -14250.218} C_VEL
LIN {X 0,Y 461.633,Z 389.986,A -85,B 0,C 180,E1 -14251.104,E2 -14251.104} C_VEL
LIN {X 0,Y 463.272,Z 391.839,A -85,B 0,C 180,E1 -14251.511,E2 -14251.511} C_VEL
LIN {X 0,Y 467.173,Z 396.479,A -85,B 0,C 180,E1 -14252.458,E2 -14252.458} C_VEL
LIN {X 0,Y 476.963,Z 409.138,A -85,B 0,C 180,E1 -14254.692,E2 -14254.692} C_VEL
LIN {X 0,Y 484.786,Z 419.482,A -85,B 0,C 180,E1 -14256.332,E2 -14256.332} C_VEL
LIN {X 0,Y 496.615,Z 435.891,A -85,B 0,C 180,E1 -14258.621,E2 -14258.621} C_VEL
LIN {X 0,Y 508.771,Z 454.299,A -85,B 0,C 180,E1 -14260.785,E2 -14260.785} C_VEL
LIN {X 0,Y 513.368,Z 462.385,A -85,B 0,C 180,E1 -14261.576,E2 -14261.576} C_VEL
LIN {X 0,Y 502.369,Z 714.276,A -85,B 0,C 180,E1 -14265.407,E2 -14265.407} C_VEL
LIN {X 0,Y 500.529,Z 749.674,A -85,B 0,C 180,E1 -14265.989,E2 -14265.989} C_VEL
LIN {X 0,Y 498.414,Z 772.695,A -85,B 0,C 180,E1 -14266.534,E2 -14266.534} C_VEL
LIN {X 0,Y 495.629,Z 796.424,A -85,B 0,C 180,E1 -14267.272,E2 -14267.272} C_VEL
LIN {X 0,Y 492.352,Z 818.328,A -85,B 0,C 180,E1 -14268.154,E2 -14268.154} C_VEL
LIN {X 0,Y 488.749,Z 839.499,A -85,B 0,C 180,E1 -14269.184,E2 -14269.184} C_VEL
LIN {X 0,Y 484.276,Z 862.069,A -85,B 0,C 180,E1 -14270.511,E2 -14270.511} C_VEL
LIN {X 0,Y 480.234,Z 880.63,A -85,B 0,C 180,E1 -14271.802,E2 -14271.802} C_VEL
LIN {X 0,Y 475.211,Z 901.882,A -85,B 0,C 180,E1 -14273.53,E2 -14273.53} C_VEL
LIN {X 0,Y 470.686,Z 919.635,A -85,B 0,C 180,E1 -14275.223,E2 -14275.223} C_VEL
LIN {X 0,Y 465.808,Z 938.147,A -85,B 0,C 180,E1 -14277.253,E2 -14277.253} C_VEL
LIN {X 0,Y 461.166,Z 954.845,A -85,B 0,C 180,E1 -14279.403,E2 -14279.403} C_VEL
LIN {X 0,Y 456.779,Z 970.943,A -85,B 0,C 180,E1 -14281.782,E2 -14281.782} C_VEL
LIN {X 0,Y 452.707,Z 985.688,A -85,B 0,C 180,E1 -14284.348,E2 -14284.348} C_VEL
LIN {X 0,Y 449.323,Z 998.642,A -85,B 0,C 180,E1 -14286.942,E2 -14286.942} C_VEL
LIN {X 0,Y 446.265,Z 1010.913,A -85,B 0,C 180,E1 -14289.852,E2 -14289.852} C_VEL
LIN {X 0,Y 444.102,Z 1020.716,A -85,B 0,C 180,E1 -14292.576,E2 -14292.576} C_VEL
LIN {X 0,Y 442.278,Z 1030.14,A -85,B 0,C 180,E1 -14295.734,E2 -14295.734} C_VEL
LIN {X 0,Y 441.394,Z 1035.6,A -85,B 0,C 180,E1 -14297.926,E2 -14297.926} C_VEL
LIN {X 0,Y 440.111,Z 1037.859,A -85,B 0,C 180,E1 -14298.88,E2 -14298.88} C_VEL
LIN {X 0,Y 433.155,Z 1043.266,A -85,B 0,C 180,E1 -14301.502,E2 -14301.502} C_VEL
LIN {X 0,Y 432.383,Z 1044.478,A -85,B 0,C 180,E1 -14302.289,E2 -14302.289} C_VEL
LIN {X 0,Y 432.089,Z 1048.284,A -85,B 0,C 180,E1 -14305.221,E2 -14305.221} C_VEL
LIN {X 0,Y 431.976,Z 1050.837,A -85,B 0,C 180,E1 -14308.408,E2 -14308.408} C_VEL
LIN {X 0,Y 431.951,Z 1051.8,A -85,B 0,C 180,E1 -14311.061,E2 -14311.061} C_VEL
LIN {X 0,Y 431.954,Z 1051.698,A -85,B 0,C 180,E1 -14313.897,E2 -14313.897} C_VEL
LIN {X 0,Y 432.022,Z 1050.014,A -85,B 0,C 180,E1 -14317.18,E2 -14317.18} C_VEL
LIN {X 0,Y 432.173,Z 1047.424,A -85,B 0,C 180,E1 -14319.858,E2 -14319.858} C_VEL
LIN {X 0,Y 432.574,Z 1043.346,A -85,B 0,C 180,E1 -14322.821,E2 -14322.821} C_VEL
LIN {X 0,Y 433.432,Z 1037.204,A -85,B 0,C 180,E1 -14326.071,E2 -14326.071} C_VEL
LIN {X 0,Y 434.663,Z 1030.406,A -85,B 0,C 180,E1 -14328.926,E2 -14328.926} C_VEL
LIN {X 0,Y 436.848,Z 1020.417,A -85,B 0,C 180,E1 -14332.331,E2 -14332.331} C_VEL
LIN {X 0,Y 439.249,Z 1010.8,A -85,B 0,C 180,E1 -14335.05,E2 -14335.05} C_VEL
LIN {X 0,Y 442.83,Z 997.813,A -85,B 0,C 180,E1 -14338.159,E2 -14338.159} C_VEL
LIN {X 0,Y 446.49,Z 985.27,A -85,B 0,C 180,E1 -14340.703,E2 -14340.703} C_VEL
LIN {X 0,Y 451.054,Z 970.157,A -85,B 0,C 180,E1 -14343.351,E2 -14343.351} C_VEL
LIN {X 0,Y 455.508,Z 955.338,A -85,B 0,C 180,E1 -14345.57,E2 -14345.57} C_VEL
LIN {X 0,Y 460.715,Z 938.153,A -85,B 0,C 180,E1 -14347.815,E2 -14347.815} C_VEL
LIN {X 0,Y 465.91,Z 919.972,A -85,B 0,C 180,E1 -14349.829,E2 -14349.829} C_VEL
LIN {X 0,Y 470.913,Z 901.887,A -85,B 0,C 180,E1 -14351.57,E2 -14351.57} C_VEL
